(****************************************************************Mode 21 : Mode alerte préparateur****************************************************************)
Mode_21 := Numero_Mode = 21 AND Enable;
TON_Mode21(IN:=(Mode_21 AND NOT Fin_Action), PT:= T#10s);
IF(Mode_21)
	THEN
	(*Gestion du texte du mode*)
	Out_Texte_FR := 'ALERTE PREPARATEUR';
	Out_Texte_ENG := 'PREPARATOR ALERT';

	(*Initialisation des actionneurs non utilisés*)
	Cmd_Douche := FALSE;
	Cmd_Lavabo := FALSE;
	Cmd_Douchette := FALSE;
	Cmd_NEP := FALSE;
	Cmd_Electrovanne_Douche := FALSE;
	Cmd_Electrovanne_Lavabo := FALSE;
	Cmd_Verin_WC_GV := FALSE;
	Cmd_Verin_WC_PV := FALSE;
END_IF;

(****************************************************************Mode 22 : Mode alerte évaluateur****************************************************************)
Mode_22 := Numero_Mode = 22 AND Enable;
TON_Mode22(IN:=(Mode_22 AND NOT Fin_Action), PT:= T#10s);
IF(Mode_22)
	THEN
	(*Gestion du texte du mode*)
	Out_Texte_FR := 'ALERTE EVALUATEUR';
	Out_Texte_ENG := 'EVALUATOR ALERT';

	(*Initialisation des actionneurs non utilisés*)
	Cmd_Douche := FALSE;
	Cmd_Lavabo := FALSE;
	Cmd_Douchette := FALSE;
	Cmd_NEP := FALSE;
	Cmd_Electrovanne_Douche := FALSE;
	Cmd_Electrovanne_Lavabo := FALSE;
	Cmd_Verin_WC_GV := FALSE;
	Cmd_Verin_WC_PV := FALSE;
END_IF;

(****************************************************************Mode 23 : Mode évaluation (sans moteur bypass)****************************************************************)
Mode_23 := Numero_Mode = 23 AND Enable;
F_TRIG_Texte23(CLK:= (Valid_Texte AND Mode_23));
IF(Mode_23)
	THEN
	(*Gestion du texte du mode*)
	Out_Texte_FR := 'EVALUATION';
	Out_Texte_ENG := 'EVALUATION';

	(*Gestion des lectures consignes du mode*)
	Out_Debit_Souf 			:= Cons_Deb_Soufflage;
	Out_Debit_Ext 			:= Cons_Deb_Extraction;
	Out_Temp_Eau 			:= Cons_Temperature_Eau;

	(*Initialisation des actionneurs non utilisés*)
	Cmd_Douche := FALSE;
	Cmd_Lavabo := FALSE;
	Cmd_Douchette := FALSE;
	Cmd_NEP := FALSE;
	Cmd_Vidange_Douche := FALSE;
	//Cmd_Vidange_Lavabo := FALSE;
	Cmd_Electrovanne_Douche := FALSE;
	Cmd_Electrovanne_Lavabo := FALSE;
	Cmd_Prise := FALSE;
	Cmd_Verin_WC_GV := FALSE;
	Cmd_Verin_WC_PV := FALSE;
END_IF;

(****************************************************************Mode 24 : Mode évaluation (avec moteur bypass)****************************************************************)
Mode_24 := Numero_Mode = 24 AND Enable;
F_TRIG_Texte24(CLK:= (Valid_Texte AND Mode_24));
IF(Mode_24)
	THEN
	(*Gestion du texte du mode*)
	Out_Texte_FR := 'EVALUATION AVEC AIR';
	Out_Texte_ENG := 'EVALUATION WITH AIR FLOW';

	(*Gestion des lectures consignes du mode*)
	Out_Debit_Souf 			:= 0.0;
	Out_Debit_Ext 			:= 0.0;
	Out_Temp_Eau 			:= Cons_Temperature_Eau;
	Out_Cons_Moteur_ByPass := REAL_TO_INT(Cons_Moteur_ByPass);

	(*Initialisation des actionneurs non utilisés*)
	Cmd_Douche := FALSE;
	Cmd_Lavabo := FALSE;
	Cmd_Douchette := FALSE;
	Cmd_NEP := FALSE;
	Cmd_Vidange_Douche := FALSE;
	Cmd_Vidange_Lavabo := FALSE;
	Cmd_Electrovanne_Douche := FALSE;
	Cmd_Electrovanne_Lavabo := FALSE;
	Cmd_Prise := FALSE;
	Cmd_Verin_WC_GV := FALSE;
	Cmd_Verin_WC_PV := FALSE;
	ELSE
	Out_Cons_Moteur_ByPass := 0;
END_IF;

(****************************************************************Mode 25 : Mode Mise en condition****************************************************************)
Mode_25 := Numero_Mode = 25 AND Enable;
F_TRIG_Mode25(CLK:= ((Valid_Texte OR R_TRIG_Valide_TempHygro.Q) AND Mode_25));
IF(Mode_25  AND NOT Fin_Action)
THEN
	(*Gestion du texte du mode*)
	Out_Texte_FR := 'MISE EN CONDITION';
	Out_Texte_ENG := 'CONDITIONING BOOTH';
	
	(*Initialisation des actionneurs non utilisés*)
	Cmd_Douche := FALSE;
	Cmd_Lavabo := FALSE;
	Cmd_Douchette := FALSE;
	Cmd_NEP := FALSE;
	Cmd_Vidange_Douche := FALSE;
	//Cmd_Vidange_Lavabo := FALSE;
	Cmd_Electrovanne_Douche := FALSE;
	Cmd_Electrovanne_Lavabo := FALSE;
	Cmd_Prise := FALSE;
	Cmd_Verin_WC_GV := FALSE;
	Cmd_Verin_WC_PV := FALSE;
	
	(*Gestion des lectures consignes du mode*)
	Out_Debit_Souf 			:= Cons_Deb_Soufflage;
	Out_Debit_Ext 			:= Cons_Deb_Extraction;
	Out_Para_11				:= Cons_Para_11;
	Out_Para_12				:= Cons_Para_12;
END_IF;
(*Validation de la régulation de la température pour passer en mode 13*)
(*Température*)
IF ((S_Ecart_Regul_PID_Temp >= 0.0) AND (S_Ecart_Regul_PID_Temp <= 2.0) AND Mode_25) THEN Temp_Ok := TRUE; ELSE Temp_Ok := FALSE; END_IF;
TON_Temp_Ok(IN:= Temp_Ok, PT:= T#15M);
(*Hygrométrie*)
IF ((S_Ecart_Regul_PID_Hygro >= 0.0) AND (S_Ecart_Regul_PID_Hygro <= 5.0) AND Mode_25) THEN Hygro_Ok := TRUE; ELSE Hygro_Ok := FALSE; END_IF;
TON_Hygro_Ok(IN:= Hygro_Ok, PT:= T#15M);
Validation_Temp_Hygro := TON_Temp_Ok.Q AND TON_Hygro_Ok.Q;
R_TRIG_Valide_TempHygro(CLK:= Validation_Temp_Hygro);

(*TP_RAZ_Mode25(IN:= Validation_Temp_Hygro, PT:= T#1s);
Validation_Temp_Hygro := (SEL(Validation_Temp_Hygro, Validation_Temp_Hygro, FALSE) OR TP_RAZ_Mode25.Q);*)

(****************************************************************Mode 26 : Mode chasse d'eau petit volume****************************************************************)
Mode_26 := Numero_Mode = 26 AND Enable;
IF(Mode_26 AND NOT Fin_Action)
	THEN
	(*Gestion du texte*)
	Out_Texte_FR := 'CHASSE D EAU PETIT VOLUME';
	Out_Texte_ENG := 'SMALL VOLUME TOILET FLUSH';

	(*Gestion du décompte de la temporisation du mode*)
	Out_Restant_Seconde := TON_Mode26.Seconde_Restant;
	Out_Restant_Minute := TON_Mode26.Minute_Restant;
	Out_Restant_Heure := TON_Mode26.Heure_Restant;

	(*Démarrage du premier cycle de chasse avant la temporisation*)
	R_TRIG_Cpt_Chasse_PV(CLK:= (Mode_26));

	(*Comptage du nombre de cycle x*)
	IF (TON_Mode26.Q OR R_TRIG_Cpt_Chasse_PV.Q)
		THEN
		Cpt_Chasse_PV := Cpt_Chasse_PV + 1;
		Restart_Chasse_PV := TRUE;
	END_IF;

	(*Initialisation des actionneurs non utilisés*)
	Cmd_Douche := FALSE;
	Cmd_Lavabo := FALSE;
	Cmd_Douchette := FALSE;
	Cmd_NEP := FALSE;
	Cmd_Electrovanne_Douche := FALSE;
	Cmd_Electrovanne_Lavabo := FALSE;
	Cmd_Prise := FALSE;
	Cmd_Verin_WC_GV := FALSE;
END_IF;
(*************************************Temporisation du décompte du mode*************************************)
TON_Mode26(
	Enable:= ((Mode_26 OR Comande_Pause OR Tp_ChasseEau_PV.Q) AND NOT Restart_Chasse_PV),
	Pause:= Comande_Pause OR Tp_ChasseEau_PV.Q,
	In_Cons_Seconde:= Tempo_Transition_Seconde,
	In_Cons_Minute:= Tempo_Transition_Minute,
	In_Cons_Heure:= Tempo_Transition_Heure);
Restart_Chasse_PV := FALSE;
(*Commande de la chasse d'eau pendant x secondes*)
Tp_ChasseEau_PV(IN:= TON_Mode26.Q OR R_TRIG_Cpt_Chasse_PV.Q, PT:= T#2s);
IF (Tp_ChasseEau_PV.Q AND Mode_26) THEN Cmd_Verin_WC_PV := TRUE; ELSE Cmd_Verin_WC_PV := FALSE; END_IF;
(*FIn du mode quand le nombre de cycle est atteint*)
IF ((Cpt_Chasse_PV >= Cons_Nbre_Chasse) AND Mode_26 AND NOT Tp_ChasseEau_PV.Q)
	THEN Etp_Suiv_ChasseEau_PV := TRUE; Cpt_Chasse_PV := 0.0;
	ELSE Etp_Suiv_ChasseEau_PV := FALSE; END_IF;
	
(****************************************************************Mode 27 : Mode lavage NEP ****************************************************************)
Mode_27 := Numero_Mode = 27 AND Enable;
IF(Mode_27  AND NOT Fin_Action)
	THEN
	(*Gestion du texte*)
	IF(E_Vanne_Vidange_Douche_Ouv)
		THEN
		Out_Texte_FR := 'LAVAGE NEP';
		Out_Texte_ENG := 'CLEANING';
		ELSE
		Out_Texte_FR := 'LAVAGE NEP - OUVERTURE BONDE';
		Out_Texte_ENG :=  'CLEANING - OPENING DRAIN';
	END_IF;
	IF(RS_Fin_Mode_27.Q1)
		THEN
		Out_Texte_FR := 'LAVAGE NEP - ARRET LAVAGE';
		Out_Texte_ENG := 'CLEANING - STOPING CLEANING';
	END_IF;

	(*Gestion de la commande de la NEP et de la vidange*)
	Cmd_Vidange_Douche := TRUE;
	
	IF( RS_Fin_Mode_27.Q1)
		THEN
		Out_Restant_Seconde := 0.0;
		Out_Restant_Minute := 0.0;
		Out_Restant_Heure := 0.0;
		Cmd_NEP := FALSE;
		ELSE
		IF(E_Vanne_Vidange_Douche_Ouv)
			THEN
			Cmd_NEP := TRUE;
			ELSE
			Cmd_NEP := FALSE;
		END_IF;
	END_IF;

	(*Gestion de la commande pause*)
	IF(Comande_Pause)
		THEN
		Cmd_NEP := FALSE;
	END_IF;

	(*Gestion du décompte de la temporisation du mode*)
	Out_Restant_Seconde := TON_Mode27.Seconde_Restant;
	Out_Restant_Minute := TON_Mode27.Minute_Restant;
	Out_Restant_Heure := TON_Mode27.Heure_Restant;

	(*Gestion des lectures consignes du mode*)
	Out_Debit_Souf 			:= Cons_Deb_Soufflage;
	Out_Debit_Ext 			:= Cons_Deb_Extraction;
	(*Out_Temp_Eau 			:= Cons_Temperature_Eau;*)

	(*Initialisation des actionneurs non utilisés*)
	Cmd_Douche := FALSE;
	Cmd_Lavabo := FALSE;
	Cmd_Douchette := FALSE;
	Cmd_Vidange_Lavabo := FALSE;
	Cmd_Electrovanne_Douche := FALSE;
	Cmd_Electrovanne_Lavabo := FALSE;
	Cmd_Prise := FALSE;
	Cmd_Verin_WC_GV := FALSE;
	Cmd_Verin_WC_PV := FALSE;
END_IF;
(*************************************Temporisation du décompte du mode*************************************)
TON_Mode27(
Enable:= (Mode_27 AND ((E_Vanne_Vidange_Douche_Ouv AND E_Vanne_Alim_NEP_Ouv) OR Comande_Pause)),
Pause:= Comande_Pause,
In_Cons_Seconde:= Tempo_Transition_Seconde,
In_Cons_Minute:= Tempo_Transition_Minute,
In_Cons_Heure:= Tempo_Transition_Heure);

(*Activation de la fin du mode*)
RS_Fin_Mode_27(SET:= TON_Mode27.Q, RESET1:= NOT Mode_27);
IF( RS_Fin_Mode_27.Q1)
	THEN
	Out_Restant_Seconde := 0.0;
	Out_Restant_Minute := 0.0;
	Out_Restant_Heure := 0.0;
END_IF;

(****************************************************************Mode 28 : Mode en fonctionnement****************************************************************)
Mode_28 := Numero_Mode = 28 AND Enable;
F_TRIG_Mode28(CLK:= (Valid_Texte AND Mode_28));
IF(Mode_28 AND NOT Fin_Action)
THEN
	(*Gestion du texte du mode*)
	Out_Texte_FR := 'CABINE EN CONDITION';
	Out_Texte_ENG := 'BOOTH IN CONDITION';
	
	(*Initialisation des actionneurs non utilisés*)
	Cmd_Douche := FALSE;
	Cmd_Lavabo := FALSE;
	Cmd_Douchette := FALSE;
	Cmd_NEP := FALSE;
	Cmd_Vidange_Douche := FALSE;
	//Cmd_Vidange_Lavabo := FALSE;
	Cmd_Electrovanne_Douche := FALSE;
	Cmd_Electrovanne_Lavabo := FALSE;
	Cmd_Prise := FALSE;
	Cmd_Verin_WC_GV := FALSE;
	Cmd_Verin_WC_PV := FALSE;
	
	(*Gestion des lectures consignes du mode*)
	Out_Debit_Souf 			:= Cons_Deb_Soufflage;
	Out_Debit_Ext 			:= Cons_Deb_Extraction;
	Out_Para_11				:= Cons_Para_11;
	Out_Para_12				:= Cons_Para_12;
END_IF;

(****************************************************************Mode 30 à 59 : Mode Texte 1 à 30****************************************************************)
Mode_30 := ((Numero_Mode >= 30) AND (Numero_Mode <= 59)) AND Enable;
F_TRIG_Texte30(CLK:= (Valid_Texte AND Mode_30));
IF(Mode_30)
THEN
	(*Gestion du texte du mode*)
	Out_Texte_FR := Tab_Mode_Texte[1, (REAL_TO_INT(Numero_Mode))];
	Out_Texte_ENG := Tab_Mode_Texte[2, (REAL_TO_INT(Numero_Mode))];

	(*Initialisation des actionneurs non utilisés*)
	Cmd_Douche := FALSE;
	Cmd_Lavabo := FALSE;
	Cmd_Douchette := FALSE;
	Cmd_NEP := FALSE;
	Cmd_Electrovanne_Douche := FALSE;
	Cmd_Electrovanne_Lavabo := FALSE;
	Cmd_Verin_WC_GV := FALSE;
	Cmd_Verin_WC_PV := FALSE;
END_IF;

(****************************************************************Mode 99 : Mode END****************************************************************)
IF(Numero_Mode = 99 AND Enable)
	THEN
	Mode_END := TRUE;
	ELSE
	Mode_END := FALSE;
END_IF;

(****************************************************************Sécurité de débordement de la douche****************************************************************)
(*Sécurité douche version temporisation pour le mode 2*)
Temp_Secu_Douche := TO_TIME((TO_DINT(Temp_Secu_Debord_Douche + 5)) * 1000);
Temp_Secu_Debord_Douche_Int := (Temp_Secu_Debord_Douche); (*Pour lecture IHM*)
TON_Secu_Douche(IN:= ((Mode_2 AND (Cmd_Douche OR Cmd_Electrovanne_Douche)) AND NOT Cmd_Vidange_Douche), PT:= Temp_Secu_Douche);
IF(TON_Secu_Douche.Q)
	THEN
	Securite_Debord_Douche := TRUE;
	Cmd_Douche := FALSE;
	ELSE
	Securite_Debord_Douche := FALSE;
END_IF;

(*Sécurité lavabo version temporisation pour le mode 5*)
Temp_Secu_Lavabo := TO_TIME((TO_DINT(Temp_Secu_Debord_Lavabo + 5)) * 1000);
Temp_Secu_Debord_Lavabo_Int := (Temp_Secu_Debord_Lavabo); (*Pour lecture IHM*)
TON_Secu_Lavabo(IN:= ((Mode_5 AND (Cmd_Lavabo OR Cmd_Electrovanne_Lavabo)) AND NOT Cmd_Vidange_Lavabo) , PT:= Temp_Secu_Lavabo);
IF(TON_Secu_Lavabo.Q)
	THEN
	Securite_Debord_Lavabo := TRUE;
	Cmd_Lavabo := FALSE;
	ELSE
	Securite_Debord_Lavabo := FALSE;
END_IF;

(*Sécurité douche version débitmétre pour le mode 13*)
Secu_Volume_Douche := (((Cmd_Electrovanne_Douche AND Option_Debitmetre_Douche) AND NOT Cmd_Vidange_Douche)
						AND (Out_Volume_Eau_Douche > Volume_Secu_Debord_Douche + 0.5));
IF(Mode_13 AND Secu_Volume_Douche)
	THEN
	Securite_Debord_Douche_Debit := TRUE;
	Cmd_Electrovanne_Douche := FALSE;
	ELSE
	Securite_Debord_Douche_Debit := FALSE;
END_IF;

(*Sécurité lavabo version débitmétre pour le mode 15*)
Secu_Volume_Lavabo := (((Cmd_Electrovanne_Lavabo AND Option_Debitmetre_Lavabo) AND NOT Cmd_Vidange_Lavabo)
						AND (Out_Volume_Eau_Lavabo > Volume_Secu_Debord_Lavabo + 0.5));
IF(Mode_15 AND Secu_Volume_Lavabo)
	THEN
	Securite_Debord_Lavabo_Debit := TRUE;
	Cmd_Electrovanne_Lavabo := FALSE;
	ELSE
	Securite_Debord_Lavabo_Debit := FALSE;
END_IF;

(****************************************************************Gestion initialisation des variables****************************************************************)
IF(Numero_Mode = 0 OR Numero_Etape = 0)
	THEN
	(*Initialisation des actionneurs*)
	Cmd_Douche := FALSE;
	Cmd_Lavabo := FALSE;
	Cmd_Douchette := FALSE;
	Cmd_NEP := FALSE;
	Cmd_Vidange_Douche := FALSE;
	Cmd_Vidange_Lavabo := FALSE;
	Cmd_Electrovanne_Douche := FALSE;
	Cmd_Electrovanne_Lavabo := FALSE;
	Cmd_Prise := FALSE;
	Cmd_Verin_WC_GV := FALSE;
	Cmd_Verin_WC_PV := FALSE;

	Out_Restant_Seconde := 0.0;
	Out_Restant_Minute := 0.0;
	Out_Restant_Heure := 0.0;

	Out_Volume_Eau_Douche := 0.0;
	Out_Volume_Eau_Lavabo := 0.0;
	Out_Debit_Souf := 0.0;
	Out_Debit_Ext := 0.0;
	Out_Temp_Eau := 0.0;
	Out_Cons_V3V_Eau_Mitig := 0.0;
	Cpt_Chasse_GV := 0.0;
	Restart_Chasse_GV := FALSE;
	Etp_Suiv_ChasseEau_GV := FALSE;
	Cpt_Chasse_PV := 0.0;
	Restart_Chasse_PV := FALSE;
	Etp_Suiv_ChasseEau_PV := FALSE;
	Out_Para_11 := 0.0;
	Out_Para_12 := 0.0;
	Out_Para_13 := 0.0;
	Out_Para_14 := 0.0;
	Out_Para_15 := 0.0;

	Out_Texte_FR := '';
	Out_Texte_ENG := '';

	R_TRIG_Mode12(CLK := FALSE);
	Integr_Vol_Eau_Mode12(Enable:= FALSE);
	R_TRIG_Mode13(CLK := FALSE);
	Integr_Vol_Eau_Mode13(Enable:= FALSE);
	R_TRIG_Mode14(CLK := FALSE);
	Integr_Vol_Eau_Mode14(Enable:= FALSE);
	R_TRIG_Mode15(CLK := FALSE);
	Integr_Vol_Eau_Mode15(Enable:= FALSE);
	R_TRIG_Cpt_Chasse_GV(CLK:= FALSE);
	R_TRIG_Cpt_Chasse_PV(CLK:= FALSE);

	TON_Temp_Ok(IN:= FALSE);
	TON_Hygro_Ok(IN:= FALSE);
	TP_RAZ_Mode25(IN:= FALSE);
	F_TRIG_Mode25(CLK:= FALSE);
	F_TRIG_Mode28(CLK:= FALSE);
	Temp_Ok := FALSE;
	Hygro_Ok := FALSE;
	Validation_Temp_Hygro := FALSE;
END_IF;

(****************************************************************Gestion du passage entre chaque mode****************************************************************)
				(*Mode temporisé*)
Fin_Action := 		(RS_Fin_Mode_1.Q1 AND (E_Vanne_Alim_Douche_Ferm OR Option_Debitmetre_Douche)) (*Mode douche avec vidange*)
				OR ((RS_Fin_Mode_2.Q1 AND (E_Vanne_Alim_Douche_Ferm OR Option_Debitmetre_Douche) OR Securite_Debord_Douche)) (*Mode douche sans vidange*)
				OR (RS_Fin_Mode_4.Q1 AND (E_Vanne_Alim_Lavabo_Ferm OR Option_Debitmetre_Lavabo)) (*Mode lavabo avec vidange*)
				OR ((RS_Fin_Mode_5.Q1 AND (E_Vanne_Alim_Lavabo_Ferm OR Option_Debitmetre_Lavabo) OR Securite_Debord_Lavabo)) (*Mode lavabo sans vidange*)
				OR (RS_Fin_Mode_7.Q1) (*Mode vidange*)
				OR (RS_Fin_Mode_18.Q1 AND E_Vanne_Alim_NEP_Ferm) (*Mode lavage eau chaude*)
				OR (RS_Fin_Mode_19.Q1 AND E_Vanne_Alim_NEP_Ferm) (*Mode lavage eau froide*)
				OR (RS_Fin_Mode_27.Q1 AND E_Vanne_Alim_NEP_Ferm) (*Mode lavage*)
				(*Mode Gestion volume*)
				OR R_TRIG_Mode12.Q OR R_TRIG_Mode13.Q OR R_TRIG_Mode14.Q OR R_TRIG_Mode15.Q
				 (*Gestion des modes sans validation*)
				OR TON_Mode8.Q OR TON_Mode22.Q OR TON_Mode21.Q OR TON_Mode10.Q OR TON_Mode6.Q OR TON_Mode11.Q
				(*Mode texte*)
				OR F_TRIG_Texte3.Q OR F_TRIG_Texte23.Q OR F_TRIG_Texte30.Q OR F_TRIG_Texte16.Q OR F_TRIG_Texte17.Q OR F_TRIG_Texte24.Q
				(*Mode chasse d'eau*)
				OR Etp_Suiv_ChasseEau_GV OR Etp_Suiv_ChasseEau_PV
				(*Mode pour enceintes climatiques*)
				OR F_TRIG_Mode25.Q OR F_TRIG_Mode28.Q;

END_FUNCTION_BLOCK

// ---- POUs/Block/Cabines/Integr_Vol_Eau.TcPOU
FUNCTION_BLOCK Integr_Vol_Eau
VAR_INPUT
	Enable :BOOL;
	Mes_Debit_Eau :REAL; (*Mesure débit en l/min*)
END_VAR
VAR_OUTPUT
	Volume_Eau :REAL; (*Volume d'eau en Litre*)
END_VAR
VAR
	TON_Inc: TON;
	R_TRIG_1	:R_TRIG;
	R_TRIG_Inc: R_TRIG;
	TOP_INTEGRATION	:BOOL;
	Reset	:BOOL;

	FlowRate_MPS :REAL; (*Debit d'eau en l/s*)
	TimeElapsed :TIME; (*Temps écoulé depuis la dernière mesur*)
END_VAR

(*Comptage des secondes*)
TON_Inc(IN:= (NOT TOP_INTEGRATION AND NOT Reset), PT:= T#1s, Q=> TOP_INTEGRATION );
R_TRIG_Inc(CLK:= TOP_INTEGRATION);

R_TRIG_1(CLK:=TOP_INTEGRATION);
Reset := NOT Enable;

(*Convertion du débit d'eau l/min en l/s*)
FlowRate_MPS := Mes_Debit_Eau / 60.0;

(*Condition d'activation : mettre la variable Enbale à TRUE pour exécuter le calcul*)
IF (TOP_INTEGRATION)
	THEN
	Volume_Eau			:= Volume_Eau + FlowRate_MPS;
END_IF;

Volume_Eau:=SEL(Reset,(Volume_Eau),0.0);
Mes_Debit_Eau:=SEL(Reset,Mes_Debit_Eau,0.0);

END_FUNCTION_BLOCK

// ---- POUs/Block/Autres/Prise.TcPOU
FUNCTION_BLOCK Prise
VAR_INPUT
	Enable:						BOOL;
	Cmd_Prise:					BOOL;	(*Commande de la prise de courant*)
	Cabine_Seche: 				BOOL;
	Statut_Ferm_Reg_Douche:		BOOL;	(*Statut fermeture du registre de la vanne de la douche / 1 = Fermé / si registre non présence forcer la variable à TRUE*)
	Statut_Ferm_Lavabo:			BOOL;	(*Statut fermeture du registre de la vanne du lavabo / 1 = Fermé / si registre non présence forcer la variable à TRUE*)
	Statut_Electrovanne_Douche:		BOOL;
	Statut_Electrovanne_Lavabo:		BOOL;
	Statut_Def_Prise_Porte_Ouverte:		BOOL;
	Statut_Def_Discord_Alim_Prise:		BOOL;
	Statut_Defaut_Discord_PC_Cab:		BOOL;
END_VAR
VAR_OUTPUT
	STOR_Prise:			BOOL;			(*Commande de la sortie TOR de la prise*)
END_VAR
VAR
END_VAR

IF(Enable AND Cmd_Prise
	AND (Statut_Ferm_Reg_Douche OR Cabine_Seche OR Option_Debitmetre_Lavabo) AND (Statut_Ferm_Lavabo OR Cabine_Seche OR Option_Debitmetre_Lavabo)
	AND ( NOT Statut_Electrovanne_Douche OR Cabine_Seche) AND (NOT Statut_Electrovanne_Lavabo OR Cabine_Seche)
	AND NOT Statut_Def_Prise_Porte_Ouverte AND NOT Statut_Def_Discord_Alim_Prise AND NOT Statut_Defaut_Discord_PC_Cab)
	THEN
		STOR_Prise := TRUE;
	ELSE
		STOR_Prise := FALSE;
END_IF;

END_FUNCTION_BLOCK

// ---- POUs/h_Enr_Recette.TcPOU
PROGRAM h_Enr_Recette
VAR
	i: INT;
	F_TRIG_Reset: F_TRIG;
	j: INT;
	R_TRIG_Enr: R_TRIG;
END_VAR

R_TRIG_Enr(CLK:= Cmd_Enr_Recette AND NOT Mode_Cabine_Automatique AND NOT Validation_Recette_Auto AND NOT Start_Recette_Mode_Auto);
IF(R_TRIG_Enr.Q)
	THEN
	(*Transfert dans la recette à enregistrée dans le tableau recette automatique*)
	FOR i := 1 TO 29 BY 1 DO
		Tab_Recette_Auto[Numero_Recette_Sel, i, 1] := Tab_Enr_Recette[0, i, 1];
		Tab_Recette_Auto[Numero_Recette_Sel, i, 2] := Tab_Enr_Recette[0, i, 2];
		Tab_Recette_Auto[Numero_Recette_Sel, i, 3] := Tab_Enr_Recette[0, i, 3];
		Tab_Recette_Auto[Numero_Recette_Sel, i, 4] := Tab_Enr_Recette[0, i, 4];
		Tab_Recette_Auto[Numero_Recette_Sel, i, 5] := Tab_Enr_Recette[0, i, 5];
		Tab_Recette_Auto[Numero_Recette_Sel, i, 6] := Tab_Enr_Recette[0, i, 6];
		Tab_Recette_Auto[Numero_Recette_Sel, i, 7] := Tab_Enr_Recette[0, i, 7];
		Tab_Recette_Auto[Numero_Recette_Sel, i, 8] := Tab_Enr_Recette[0, i, 8];
		Tab_Recette_Auto[Numero_Recette_Sel, i, 9] := Tab_Enr_Recette[0, i, 9];
		Tab_Recette_Auto[Numero_Recette_Sel, i, 10] := Tab_Enr_Recette[0, i, 10];
		Tab_Recette_Auto[Numero_Recette_Sel, i, 11] := Tab_Enr_Recette[0, i, 11];
		Tab_Recette_Auto[Numero_Recette_Sel, i, 12] := Tab_Enr_Recette[0, i, 12];
		Tab_Recette_Auto[Numero_Recette_Sel, i, 13] := Tab_Enr_Recette[0, i, 13];
		Tab_Recette_Auto[Numero_Recette_Sel, i, 14] := Tab_Enr_Recette[0, i, 14];
		Tab_Recette_Auto[Numero_Recette_Sel, i, 15] := Tab_Enr_Recette[0, i, 15];
	END_FOR;
END_IF;
(*Reset du tableau sur le front descendant*)
F_TRIG_Reset(CLK:= Cmd_Enr_Recette);
IF(F_TRIG_Reset.Q)
	THEN
	FOR j := 1 TO 29 BY 1 DO
		Tab_Enr_Recette[0, j, 1] := 0;
		Tab_Enr_Recette[0, j, 2] := 0;
		Tab_Enr_Recette[0, j, 3] := 0;
		Tab_Enr_Recette[0, j, 4] := 0;
		Tab_Enr_Recette[0, j, 5] := 0;
		Tab_Enr_Recette[0, j, 6] := 0;
		Tab_Enr_Recette[0, j, 7] := 0;
		Tab_Enr_Recette[0, j, 8] := 0;
		Tab_Enr_Recette[0, j, 9] := 0;
		Tab_Enr_Recette[0, j, 10] := 0;
		Tab_Enr_Recette[0, j, 11] := 0;
		Tab_Enr_Recette[0, j, 12] := 0;
		Tab_Enr_Recette[0, j, 13] := 0;
		Tab_Enr_Recette[0, j, 14] := 0;
		Tab_Enr_Recette[0, j, 15] := 0;
	END_FOR;
	ELSE
	j := 1;
END_IF;

END_PROGRAM

// ---- POUs/i_Protocol_Auto.TcPOU
PROGRAM i_Protocol_Auto
VAR
(*Validation de la recette sélectionnée*)
	n: INT;
	i: INT;
	R_TRIG_RAZ_etape: R_TRIG;
(*initialisation des valeurs*)
	j: INT;
(*Execution de la recette en mode auto*)
	R_TRIG_Dem: R_TRIG;
	R_TRIG1: R_TRIG;
(*Gestion de la poste de ventilation*)
	F_TRIG_Fin_Post_Ventil: F_TRIG;
	TON_PV: TON;
	R_TRIG_PV: R_TRIG;
END_VAR

(*MEMSET(ADR(Tab_Nom_Recette),0,SIZEOF(Tab_Nom_Recette));
MEMSET(ADR(Tab_Mode_Texte),0,SIZEOF(Tab_Mode_Texte));*)

(************************************************************************************************************************Gestion Arrêt du grafcet*)
Mode_Arret_Auto := 	(Reset_Mode_Auto(*Fin de la recette*)
					OR ((Numero_Mode_Auto = 1) AND Mode_Auto.Mode_END) (*Fin de la recette*)
					OR (Mode_Auto.Mode_12 AND Defaut_Discord_Deb_Eau_Douche)
					OR (Mode_Auto.Mode_13 AND Defaut_Discord_Deb_Eau_Douche)
					OR (Mode_Auto.Mode_14 AND Defaut_Discord_Deb_Eau_Lavabo)
					OR (Mode_Auto.Mode_15 AND Defaut_Discord_Deb_Eau_Lavabo)
					OR Defaut_Debordement_Douche OR Defaut_Debordement_Lavabo)
					OR (Mode_Auto.Mode_4 AND Defaut_Discord_Deb_Eau_Lavabo AND Option_Debitmetre_Lavabo)
					OR (Mode_Auto.Mode_5 AND Defaut_Discord_Deb_Eau_Lavabo AND Option_Debitmetre_Lavabo)
					OR (Mode_Auto.Mode_1 AND Defaut_Discord_Deb_Eau_Douche AND Option_Debitmetre_Douche)
					OR (Mode_Auto.Mode_2 AND Defaut_Discord_Deb_Eau_Douche AND Option_Debitmetre_Douche)
					OR (RS_MEnCond.Q1 AND Defaut_Arret_Mode25 AND Option_Cabine_Climatique) //RS_MEnCond.Q1 Correspond au démarrage de la CTA durant une recette
					OR Defaut_Discord_Reg_Etanche_Ext OR Defaut_Sonde_Temp_Eau_Mitig;

(************************************************************************************************************************Validation de la recette sélectionnée*)
IF(Validation_Recette_Auto AND NOT Mode_Arret_Auto)
	THEN
	(*Remise à zéro du nombre d'étape total avant le calcul du nombre d'étape total*)
	R_TRIG_RAZ_etape(CLK:= Validation_Recette_Auto);
	IF (R_TRIG_RAZ_etape.Q) THEN Nbre_Etape_Totale := 0; END_IF;
	(*Transfert dans la recette 0 de la recettte sélectionnée*)
	FOR i := 1 TO 29 BY 1 DO
		Tab_Recette_Auto[0, i, 1] := Tab_Recette_Auto[Numero_Recette_Sel, i, 1];
		Tab_Recette_Auto[0, i, 2] := Tab_Recette_Auto[Numero_Recette_Sel, i, 2];
		Tab_Recette_Auto[0, i, 3] := Tab_Recette_Auto[Numero_Recette_Sel, i, 3];
		Tab_Recette_Auto[0, i, 4] := Tab_Recette_Auto[Numero_Recette_Sel, i, 4];
		Tab_Recette_Auto[0, i, 5] := Tab_Recette_Auto[Numero_Recette_Sel, i, 5];
		Tab_Recette_Auto[0, i, 6] := Tab_Recette_Auto[Numero_Recette_Sel, i, 6];
		Tab_Recette_Auto[0, i, 7] := Tab_Recette_Auto[Numero_Recette_Sel, i, 7];
		Tab_Recette_Auto[0, i, 8] := Tab_Recette_Auto[Numero_Recette_Sel, i, 8];
		Tab_Recette_Auto[0, i, 9] := Tab_Recette_Auto[Numero_Recette_Sel, i, 9];
		Tab_Recette_Auto[0, i, 10] := Tab_Recette_Auto[Numero_Recette_Sel, i, 10];
		Tab_Recette_Auto[0, i, 11] := Tab_Recette_Auto[Numero_Recette_Sel, i, 11];
		Tab_Recette_Auto[0, i, 12] := Tab_Recette_Auto[Numero_Recette_Sel, i, 12];
		Tab_Recette_Auto[0, i, 13] := Tab_Recette_Auto[Numero_Recette_Sel, i, 13];
		Tab_Recette_Auto[0, i, 14] := Tab_Recette_Auto[Numero_Recette_Sel, i, 14];
		Tab_Recette_Auto[0, i, 15] := Tab_Recette_Auto[Numero_Recette_Sel, i, 15];
	END_FOR;
	(*Calcul etape total*)
	FOR n := 1 TO 29 BY 1 DO
		IF(Tab_Recette_Auto[Numero_Recette_Sel, n, 1] = 99)
			THEN
			Nbre_Etape_Totale := n - 1;
			n := 29;
		END_IF;
	END_FOR;
	ELSE;
	R_TRIG_RAZ_etape(CLK:= FALSE);
	i := 0;
	n := 0;
END_IF;

(************************************************************************************************************************Démarrage du mode auto*)
IF(Mode_Cabine_Automatique AND (Numero_Mode_Auto = 0) AND NOT Mode_Arret_Auto)
	THEN
	Numero_Mode_Auto := 1;
END_IF;

(*Gestion du case du mode auto*)
CASE Numero_Mode_Auto OF
(*******************************************************************************************Etape 0 : Attente*)
0:
j:=0; (*Initlisation de la variable boucle FOR d'initialisation*)
Mode_Auto(
	Enable:= 					(FALSE),
	Numero_Etape:= 				Numero_Etape_Actuel);

(*******************************************************************************************Etape 1 :Execution de la recette en mode auto*)
1:
R_TRIG_Dem(CLK:= (Numero_Mode_Auto = 1));
(*Démarrage de l'étape 1 de la recette*)
IF(R_TRIG_Dem.Q)
	THEN
	Numero_Etape_Actuel := Numero_Etape_Actuel + 1;
END_IF;

(*Bloc fontion recette*)
Mode_Auto(
	Enable:= 					(Numero_Mode_Auto = 1),
	Numero_Etape:= 				Numero_Etape_Actuel,
	Numero_Mode:= 				Tab_Recette_Auto[0, LIMIT(1,Numero_Etape_Actuel,30), 1],
	Tempo_Transition_seconde:=	Tab_Recette_Auto[0, LIMIT(1,Numero_Etape_Actuel,30), 2],
	Tempo_Transition_Minute:=	Tab_Recette_Auto[0, LIMIT(1,Numero_Etape_Actuel,30), 3],
	Tempo_Transition_Heure:= 	Tab_Recette_Auto[0, LIMIT(1,Numero_Etape_Actuel,30), 4],
	Cons_Volume_Eau_Douche:= 	Tab_Recette_Auto[0, LIMIT(1,Numero_Etape_Actuel,30), 6],
	Cons_Volume_Eau_Lavabo:=	Tab_Recette_Auto[0, LIMIT(1,Numero_Etape_Actuel,30), 6],
	Cons_Deb_Soufflage:= 		Tab_Recette_Auto[0, LIMIT(1,Numero_Etape_Actuel,30), 7],
	Cons_Deb_Extraction:=		Tab_Recette_Auto[0, LIMIT(1,Numero_Etape_Actuel,30), 8],
	Cons_Temperature_Eau:= 		Tab_Recette_Auto[0, LIMIT(1,Numero_Etape_Actuel,30), 9],
	Cons_Nbre_Chasse:= 			Tab_Recette_Auto[0, LIMIT(1,Numero_Etape_Actuel,30), 10],
	Cons_Para_11:= 				Tab_Recette_Auto[0, LIMIT(1,Numero_Etape_Actuel,30), 11],
	Cons_Para_12:= 				Tab_Recette_Auto[0, LIMIT(1,Numero_Etape_Actuel,30), 12],
	Cons_Para_13:= 				Tab_Recette_Auto[0, LIMIT(1,Numero_Etape_Actuel,30), 13],
	Cons_Para_14:= 				Tab_Recette_Auto[0, LIMIT(1,Numero_Etape_Actuel,30), 14],
	Cons_Para_15:= 				Tab_Recette_Auto[0, LIMIT(1,Numero_Etape_Actuel,30), 15],);

(*Lecture des consignes actuel en cours de fonctionnement pour chaque étape (Valeurs en entrées du bloc Mode)*)
Numero_Mode_Actuel 				:= (Mode_Auto.Numero_Mode);
Tempo_Transition_seconde_Actuel := (Mode_Auto.Tempo_Transition_seconde);
Tempo_Transition_Minute_Actuel 	:= (Mode_Auto.Tempo_Transition_Minute);
Tempo_Transition_Heure_Actuel 	:= (Mode_Auto.Tempo_Transition_Heure);
Cons_Volume_Eau_Douche_Actuel 	:= (Mode_Auto.Cons_Volume_Eau_Douche);
Cons_Volume_Eau_Lavabo_Actuel	:= (Mode_Auto.Cons_Volume_Eau_Lavabo);
Cons_Deb_Soufflage_Actuel 		:= (Mode_Auto.Cons_Deb_Soufflage);
Cons_Deb_Extraction_Actuel 		:= (Mode_Auto.Cons_Deb_Extraction);
Cons_Temperature_Eau_Actuel 	:= (Mode_Auto.Cons_Temperature_Eau);
Cons_Para_Nbre_Chasse_Eau 		:= (Mode_Auto.Cons_Nbre_Chasse);
Cons_Para_11_Actuel 			:= (Mode_Auto.Cons_Para_11);
Cons_Para_12_Actuel 			:= (Mode_Auto.Cons_Para_12);
Cons_Para_13_Actuel 			:= (Mode_Auto.Cons_Para_13);
Cons_Para_14_Actuel 			:= (Mode_Auto.Cons_Para_14);
Cons_Para_15_Actuel 			:= (Mode_Auto.Cons_Para_15);

(*Lecture des consignes appliquée en cours de fonctionnement pour chaque étape (Valeurs en sorties du bloc Mode)*)
(*Affichage du texte du mode en cours*)
MEMSET(ADR(Lecture_Texte_Choisi_FR),0,SIZEOF(Lecture_Texte_Choisi_FR));
MEMSET(ADR(Lecture_Texte_Choisi_ENG),0,SIZEOF(Lecture_Texte_Choisi_ENG));
Lecture_Texte_Choisi_FR 	:= Mode_Auto.Out_Texte_FR;
Lecture_Texte_Choisi_ENG	:= Mode_Auto.Out_Texte_ENG;
(*Gestion du décompte du temps restant*)
Temp_Restant_Seconde 			:= Mode_Auto.Out_Restant_Seconde;
Temp_Restant_Minute 			:= Mode_Auto.Out_Restant_Minute;
Temp_Restant_Heure 				:= Mode_Auto.Out_Restant_Heure;
(*Gestion du décompte du nombre de chasse*)
Nbre_Chasse_Total := Mode_Auto.Cons_Nbre_Chasse;
Nbre_Chasse_EnCours := MAX(Mode_Auto.Cpt_Chasse_PV, Mode_Auto.Cpt_Chasse_GV);
(*Débit d'eau, consigne de ventilation et consigne de température d'eau*)
IF (S_Cmd_Vanne_Alim_Douche OR S_Cmd_ElectroValve_Alim_Douche) THEN
Lect_Volume_Eau_Douche 			:= LIMIT(0,(Mode_Auto.Out_Volume_Eau_Douche - Trop_Plein_Douche + Garde_Deau_Douche),150);
ELSE Lect_Volume_Eau_Douche := 0.0; END_IF;
IF (S_Cmd_Vanne_Alim_Lavabo OR S_Cmd_ElectroValve_Alim_Lavabo) THEN
Lect_Volume_Eau_Lavabo			:= LIMIT(0,(Mode_Auto.Out_Volume_Eau_Lavabo - Trop_Plein_Lavabo + Garde_Deau_Lavabo),150);
ELSE Lect_Volume_Eau_Lavabo := 0.0; END_IF;
Cons_Deb_Soufflage_Appli 		:= Mode_Auto.Out_Debit_Souf;
Cons_Deb_Extraction_Appli 		:= Mode_Auto.Out_Debit_Ext;
Cons_Temperature_Eau_Appli 		:= Mode_Auto.Out_Temp_Eau;
Cons_Para_Nbre_Chasse_Eau 		:= Mode_Auto.Cons_Nbre_Chasse;
Cons_Para_11_Appli 				:= Mode_Auto.Out_Para_11;
Cons_Para_12_Appli 				:= Mode_Auto.Out_Para_12;
Cons_Para_13_Appli 				:= Mode_Auto.Out_Para_13;
Cons_Para_14_Appli 				:= Mode_Auto.Out_Para_14;
Cons_Para_15_Appli 				:= Mode_Auto.Out_Para_15;

(*Passage à l'étape suivante*)
R_TRIG1(CLK:= Mode_Auto.Fin_Action);
IF(R_TRIG1.Q)
	THEN
	Numero_Etape_Actuel := Numero_Etape_Actuel + 1;
END_IF;

(*Fin de la recette*)
IF(Mode_Arret_Auto)
	THEN
	Numero_Mode_Auto := 3;
END_IF;

(*******************************************************************************************Gestion vérification de la poste de ventilation*)
3:
(*Attente de quelques secondes si demmande de post ventilation*)
TON_PV(IN:= (NOT Dmd_Post_Ventilation), PT:= T#1s);
R_TRIG_PV(CLK:= TON_PV.Q);
 (*Démarrage de la recette à la fin de la post ventilation*)
F_TRIG_Fin_Post_Ventil(CLK:= Dmd_Post_Ventilation);
IF(F_TRIG_Fin_Post_Ventil.Q OR R_TRIG_PV.Q)
	THEN
	Numero_Mode_Auto := 2;
END_IF;
MEMSET(ADR(Lecture_Texte_Choisi_FR),0,SIZEOF(Lecture_Texte_Choisi_FR));
MEMSET(ADR(Lecture_Texte_Choisi_ENG),0,SIZEOF(Lecture_Texte_Choisi_ENG));
IF (Dmd_Post_Ventilation) (*Affichage du texte post ventilation*)
	THEN
	Lecture_Texte_Choisi_FR 	:= 'POST VENTILATION EN COURS';
	Lecture_Texte_Choisi_ENG	:= 'POST VENTILATION IN PROCESS';
END_IF;
Mode_Auto(
	Enable:= 					FALSE,
	Numero_Etape:= 				0,
	Numero_Mode:= 				0,
	Tempo_Transition_seconde:=	0,
	Tempo_Transition_Minute:=	0,
	Tempo_Transition_Heure:= 	0,
	Cons_Volume_Eau_Douche:= 	0,
	Cons_Volume_Eau_Lavabo:=	0,
	Cons_Deb_Soufflage:= 		0,
	Cons_Deb_Extraction:=		0,
	Cons_Temperature_Eau:= 		0,
	Cons_Nbre_Chasse:= 			0,
	Cons_Para_11:= 				0,
	Cons_Para_12:= 				0,
	Cons_Para_13:= 				0,
	Cons_Para_14:= 				0,
	Cons_Para_15:= 				0);

(*******************************************************************************************Etape 2 : Initialisation des valeurs*)
2:
FOR j := 1 TO 29 BY 1 DO
	Tab_Recette_Auto[0, j, 1] := 0;
	Tab_Recette_Auto[0, j, 2] := 0;
	Tab_Recette_Auto[0, j, 3] := 0;
	Tab_Recette_Auto[0, j, 4] := 0;
	Tab_Recette_Auto[0, j, 5] := 0;
	Tab_Recette_Auto[0, j, 6] := 0;
	Tab_Recette_Auto[0, j, 7] := 0;
	Tab_Recette_Auto[0, j, 8] := 0;
	Tab_Recette_Auto[0, j, 9] := 0;
	Tab_Recette_Auto[0, j, 10] := 0;
	Tab_Recette_Auto[0, j, 11] := 0;
	Tab_Recette_Auto[0, j, 12] := 0;
	Tab_Recette_Auto[0, j, 13] := 0;
	Tab_Recette_Auto[0, j, 14] := 0;
	Tab_Recette_Auto[0, j, 15] := 0;

	Tab_Enr_Recette[0, j, 1] := 0;
	Tab_Enr_Recette[0, j, 2] := 0;
	Tab_Enr_Recette[0, j, 3] := 0;
	Tab_Enr_Recette[0, j, 4] := 0;
	Tab_Enr_Recette[0, j, 5] := 0;
	Tab_Enr_Recette[0, j, 6] := 0;
	Tab_Enr_Recette[0, j, 7] := 0;
	Tab_Enr_Recette[0, j, 8] := 0;
	Tab_Enr_Recette[0, j, 9] := 0;
	Tab_Enr_Recette[0, j, 10] := 0;
	Tab_Enr_Recette[0, j, 11] := 0;
	Tab_Enr_Recette[0, j, 12] := 0;
	Tab_Enr_Recette[0, j, 13] := 0;
	Tab_Enr_Recette[0, j, 14] := 0;
	Tab_Enr_Recette[0, j, 15] := 0;
END_FOR;

Numero_Etape_Actuel := 0;
Nbre_Etape_Totale := 0;

R_TRIG_Dem(CLK:=FALSE);
R_TRIG1(CLK:=FALSE);
F_TRIG_Fin_Post_Ventil(CLK:= FALSE);
TON_PV(IN:= (FALSE));
R_TRIG_PV(CLK:= FALSE);

Numero_Mode_Actuel 				:= 0;
Tempo_Transition_seconde_Actuel := 0;
Tempo_Transition_Minute_Actuel 	:= 0;
Tempo_Transition_Heure_Actuel 	:= 0;
Cons_Volume_Eau_Douche_Actuel 	:= 0;
Cons_Volume_Eau_Lavabo_Actuel	:= 0;
Cons_Deb_Soufflage_Actuel 		:= 0;
Cons_Deb_Extraction_Actuel 		:= 0;
Cons_Temperature_Eau_Actuel 	:= 0;
Cons_Para_Nbre_Chasse_Eau 		:= 0;
Cons_Para_11_Actuel 			:= 0;
Cons_Para_12_Actuel 			:= 0;
Cons_Para_13_Actuel 			:= 0;
Cons_Para_14_Actuel 			:= 0;
Cons_Para_15_Actuel 			:= 0;

Mode_Auto(
	Enable:= 					FALSE,
	Numero_Etape:= 				0,
	Numero_Mode:= 				0,
	Tempo_Transition_seconde:=	0,
	Tempo_Transition_Minute:=	0,
	Tempo_Transition_Heure:= 	0,
	Cons_Volume_Eau_Douche:= 	0,
	Cons_Volume_Eau_Lavabo:=	0,
	Cons_Deb_Soufflage:= 		0,
	Cons_Deb_Extraction:=		0,
	Cons_Temperature_Eau:= 		0,
	Cons_Nbre_Chasse:= 			0,
	Cons_Para_11:= 				0,
	Cons_Para_12:= 				0,
	Cons_Para_13:= 				0,
	Cons_Para_14:= 				0,
	Cons_Para_15:= 				0);

Cons_Dimmer_Auto				:= 254;
Cons_Appl_Rouge_Auto			:= 254;
Cons_Appl_Vert_Auto				:= 254;
Cons_Appl_Bleu_Auto				:= 254;
Cons_Appl_Blanc_Auto			:= 254;

MEMSET(ADR(Lecture_Texte_Choisi_FR),0,SIZEOF(Lecture_Texte_Choisi_FR));
MEMSET(ADR(Lecture_Texte_Choisi_ENG),0,SIZEOF(Lecture_Texte_Choisi_ENG));

Lecture_Texte_Choisi_FR			:= '';
Lecture_Texte_Choisi_ENG		:= '';
Temp_Restant_Seconde 			:= 0.0;
Temp_Restant_Minute 			:= 0.0;
Temp_Restant_Heure 				:= 0.0;
Lect_Volume_Eau_Douche 			:= 0.0;
Lect_Volume_Eau_Lavabo			:= 0.0;
Cons_Deb_Soufflage_Appli 		:= 0.0;
Cons_Deb_Extraction_Appli 		:= 0.0;
Cons_Temperature_Eau_Appli 		:= 0.0;
Cons_Para_Nbre_Chasse_Eau 		:= 0.0;
Cons_Para_11_Appli 				:= 0.0;
Cons_Para_12_Appli 				:= 0.0;
Cons_Para_13_Appli 				:= 0.0;
Cons_Para_14_Appli 				:= 0.0;
Cons_Para_15_Appli 				:= 0.0;

(*Retour à l'étape 0 à la fin de l'initialisation*)
Numero_Mode_Auto := 0;
END_CASE;

END_PROGRAM

// ---- POUs/j_Protocol_Manu.TcPOU
PROGRAM j_Protocol_Manu
VAR
(*Enregistrement de la recette manuel*)
	R_TRIG_Enr_Manuel: R_TRIG;
(*initialisation des valeurs*)
END_VAR

(************************************************************************************************************************Gestion Arrêt du grafcet*)
Mode_Arret_Manu := 	(Reset_Mode_Manu(*Bouton arrêt*)
					OR ((Numero_Mode_Manu = 1) AND Mode_Manu.Fin_Action) (*Fin du mode*)
					OR (Mode_Manu.Mode_12 AND Defaut_Discord_Deb_Eau_Douche)
					OR (Mode_Manu.Mode_13 AND Defaut_Discord_Deb_Eau_Douche)
					OR (Mode_Manu.Mode_14 AND Defaut_Discord_Deb_Eau_Lavabo)
					OR (Mode_Manu.Mode_15 AND Defaut_Discord_Deb_Eau_Lavabo)
					OR Defaut_Debordement_Douche OR Defaut_Debordement_Lavabo)
					OR (Mode_Manu.Mode_4 AND Defaut_Discord_Deb_Eau_Lavabo AND Option_Debitmetre_Lavabo)
					OR (Mode_Manu.Mode_5 AND Defaut_Discord_Deb_Eau_Lavabo AND Option_Debitmetre_Lavabo)
					OR (Mode_Manu.Mode_1 AND Defaut_Discord_Deb_Eau_Douche AND Option_Debitmetre_Douche)
					OR (Mode_Manu.Mode_2 AND Defaut_Discord_Deb_Eau_Douche AND Option_Debitmetre_Douche)
					OR (Mode_Auto.Mode_25 AND Defaut_Arret_Mode25 AND Option_Cabine_Climatique)
					OR Defaut_Discord_Reg_Etanche_Ext OR Defaut_Sonde_Temp_Eau_Mitig;

(************************************************************************************************************************Enregistrement de la recette manuel*)
R_TRIG_Enr_Manuel(CLK:=Mode_Cabine_Manuel);
IF(R_TRIG_Enr_Manuel.Q)
	THEN
	Tab_Enr_Mode_Manu[1] 			:= Manu_Choix_Numero_Mode;
	Tab_Enr_Mode_Manu[2] 			:= Manu_Tempo_Transition_Seconde;
	Tab_Enr_Mode_Manu[3] 			:= Manu_Tempo_Transition_Minute;
	Tab_Enr_Mode_Manu[4] 			:= Manu_Tempo_Transition_Heure;
	Tab_Enr_Mode_Manu[5] 			:= Manu_Lct_Cons_Vol_Douche;
	Tab_Enr_Mode_Manu[6] 			:= Manu_Lct_Cons_Vol_Lavabo;
	Tab_Enr_Mode_Manu[7] 			:= Manu_Cons_Deb_Soufflage;
	Tab_Enr_Mode_Manu[8] 			:= Manu_Cons_Deb_Extraction;
	Tab_Enr_Mode_Manu[9] 			:= Manu_Cons_Temp_Eau;
	Tab_Enr_Mode_Manu[10] 			:= Manu_Cons_Nbre_Chasse;
	Tab_Enr_Mode_Manu[11] 			:= Manu_Cons_Para11;
	Tab_Enr_Mode_Manu[12] 			:= Manu_Cons_Para12;
	Tab_Enr_Mode_Manu[13] 			:= Manu_Cons_Para13;
	Tab_Enr_Mode_Manu[14] 			:= Manu_Cons_Para14;
	Tab_Enr_Mode_Manu[15] 			:= Manu_Cons_Para15;
END_IF;

(************************************************************************************************************************Démarrage du mode manu*)
(*Démarrage du mode manuel à la fin de l'enregistrement*)
IF(Mode_Cabine_Manuel AND (Tab_Enr_Mode_Manu[1] <> 0))
	THEN
	Numero_Mode_Manu := 1;
END_IF;

(*Gestion du case du mode auto*)
CASE Numero_Mode_Manu OF
(*******************************************************************************************Etape 0 : Attente*)
0:
Mode_Manu(
	Enable:= 						(FALSE),
	Numero_Etape:= 					Numero_Mode_Manu);

(*******************************************************************************************Etape 1 : Execution de la recette en mode auto*)
1:
Mode_Manu(
	Enable:= 						(Numero_Mode_Manu = 1),
	Numero_Etape:= 					Numero_Mode_Manu,
	Numero_Mode:= 					Tab_Enr_Mode_Manu[1],
	Tempo_Transition_seconde:= 		Tab_Enr_Mode_Manu[2],
	Tempo_Transition_Minute:=		Tab_Enr_Mode_Manu[3],
	Tempo_Transition_Heure:= 		Tab_Enr_Mode_Manu[4],
	Cons_Volume_Eau_Douche:= 		Tab_Enr_Mode_Manu[5],
	Cons_Volume_Eau_Lavabo:=		Tab_Enr_Mode_Manu[6],
	Cons_Deb_Soufflage:=			Tab_Enr_Mode_Manu[7],
	Cons_Deb_Extraction:=			Tab_Enr_Mode_Manu[8],
	Cons_Temperature_Eau:=			Tab_Enr_Mode_Manu[9],
	Cons_Nbre_Chasse:=				Tab_Enr_Mode_Manu[10],
	Cons_Para_11:=					Tab_Enr_Mode_Manu[11],
	Cons_Para_12:= 					Tab_Enr_Mode_Manu[12],
	Cons_Para_13:=					Tab_Enr_Mode_Manu[13],
	Cons_Para_14:=					Tab_Enr_Mode_Manu[14],
	Cons_Para_15:= 					Tab_Enr_Mode_Manu[15]);

(*Lecture des consignes appliquée en cours de fonctionnement pour chaque étape (Valeurs en sorties du bloc Mode)*)
(*Affichage du texte du mode en cours*)
MEMSET(ADR(Lecture_Texte_Choisi_FR),0,SIZEOF(Lecture_Texte_Choisi_FR));
MEMSET(ADR(Lecture_Texte_Choisi_ENG),0,SIZEOF(Lecture_Texte_Choisi_ENG));
Lecture_Texte_Choisi_FR 			:= Mode_Manu.Out_Texte_FR;
Lecture_Texte_Choisi_ENG			:= Mode_Manu.Out_Texte_ENG;
(*Gestion du décompte du temps restant*)
Temp_Restant_Seconde 				:= Mode_Manu.Out_Restant_Seconde;
Temp_Restant_Minute 				:= Mode_Manu.Out_Restant_Minute;
Temp_Restant_Heure 					:= Mode_Manu.Out_Restant_Heure;
(*Gestion du décompte du nombre de chasse*)
Nbre_Chasse_Total 					:= Mode_Manu.Cons_Nbre_Chasse;
Nbre_Chasse_EnCours 				:= MAX(Mode_Manu.Cpt_Chasse_PV, Mode_Manu.Cpt_Chasse_GV);
(*Débit d'eau, consigne de ventilation et consigne de température d'eau*)
IF (S_Cmd_Vanne_Alim_Douche OR S_Cmd_ElectroValve_Alim_Douche) THEN
Lect_Volume_Eau_Douche 				:= LIMIT(0,(Mode_Manu.Out_Volume_Eau_Douche - Trop_Plein_Douche + Garde_Deau_Douche),150);
ELSE Lect_Volume_Eau_Douche 		:= 0.0; END_IF;
IF (S_Cmd_Vanne_Alim_Lavabo OR S_Cmd_ElectroValve_Alim_Lavabo) THEN
Lect_Volume_Eau_Lavabo				:= LIMIT(0,(Mode_Manu.Out_Volume_Eau_Lavabo - Trop_Plein_Lavabo + Garde_Deau_Lavabo),150);
ELSE Lect_Volume_Eau_Lavabo 		:= 0.0; END_IF;
Cons_Deb_Soufflage_Appli 			:= Mode_Manu.Out_Debit_Souf;
Cons_Deb_Extraction_Appli 			:= Mode_Manu.Out_Debit_Ext;
Cons_Temperature_Eau_Appli 			:= Mode_Manu.Out_Temp_Eau;
Cons_Para_Nbre_Chasse_Eau 			:= Mode_Manu.Cons_Nbre_Chasse;
Cons_Para_11_Appli 					:= Mode_Manu.Out_Para_11;
Cons_Para_12_Appli 					:= Mode_Manu.Out_Para_12;
Cons_Para_13_Appli 					:= Mode_Manu.Out_Para_13;
Cons_Para_14_Appli 					:= Mode_Manu.Out_Para_14;
Cons_Para_15_Appli 					:= Mode_Manu.Out_Para_15;

(*Fin du mode*)
IF(Mode_Arret_Manu)
	THEN
	Numero_Mode_Manu := 2;
END_IF;

(*******************************************************************************************Etape 2 : Initialisation des valeurs*)
2:
Tab_Enr_Mode_Manu[1] 				:= 0;
Tab_Enr_Mode_Manu[2] 				:= 0;
Tab_Enr_Mode_Manu[3] 				:= 0;
Tab_Enr_Mode_Manu[4] 				:= 0;
Tab_Enr_Mode_Manu[5] 				:= 0;
Tab_Enr_Mode_Manu[6] 				:= 0;
Tab_Enr_Mode_Manu[7] 				:= 0;
Tab_Enr_Mode_Manu[8] 				:= 0;
Tab_Enr_Mode_Manu[9] 				:= 0;
Tab_Enr_Mode_Manu[10]				:= 0;
Tab_Enr_Mode_Manu[11]				:= 0;
Tab_Enr_Mode_Manu[12]				:= 0;
Tab_Enr_Mode_Manu[13]				:= 0;
Tab_Enr_Mode_Manu[14]				:= 0;
Tab_Enr_Mode_Manu[15]				:= 0;

Mode_Manu(
	Enable:= 						FALSE,
	Numero_Etape:= 					0,
	Numero_Mode:= 					0,
	Tempo_Transition_seconde:=		0,
	Tempo_Transition_Minute:=		0,
	Tempo_Transition_Heure:= 		0,
	Cons_Volume_Eau_Douche:= 		0,
	Cons_Volume_Eau_Lavabo:=		0,
	Cons_Deb_Soufflage:= 			0,
	Cons_Deb_Extraction:=			0,
	Cons_Temperature_Eau:= 			0,
	Cons_Nbre_Chasse:= 				0,
	Cons_Para_11:= 					0,
	Cons_Para_12:= 					0,
	Cons_Para_13:= 					0,
	Cons_Para_14:= 					0,
	Cons_Para_15:= 					0);

MEMSET(ADR(Lecture_Texte_Choisi_FR),0,SIZEOF(Lecture_Texte_Choisi_FR));
MEMSET(ADR(Lecture_Texte_Choisi_ENG),0,SIZEOF(Lecture_Texte_Choisi_ENG));
Lecture_Texte_Choisi_FR				:= '';
Lecture_Texte_Choisi_ENG			:= '';
Temp_Restant_Seconde 				:= 0.0;
Temp_Restant_Minute 				:= 0.0;
Temp_Restant_Heure 					:= 0.0;
Lect_Volume_Eau_Douche 				:= 0.0;
Lect_Volume_Eau_Lavabo				:= 0.0;
Cons_Deb_Soufflage_Appli 			:= 0.0;
Cons_Deb_Extraction_Appli 			:= 0.0;
Cons_Temperature_Eau_Appli 			:= 0.0;
Cons_Para_Nbre_Chasse_Eau 			:= 0.0;
Cons_Para_11_Appli 					:= 0.0;
Cons_Para_12_Appli 					:= 0.0;
Cons_Para_13_Appli 					:= 0.0;
Cons_Para_14_Appli 					:= 0.0;
Cons_Para_15_Appli 					:= 0.0;

(*Retour à l'étape 0 à la fin de l'initialisation*)
Numero_Mode_Manu 					:= 0;
END_CASE;

END_PROGRAM

// ---- POUs/l_Cons_LED.TcPOU
PROGRAM l_Cons_LED
VAR
	Pulse_Defaut_Led_Cabine:BOOL;
	BLINK_Defaut: BLINK;
END_VAR

(*********************************Gestion du clignotement lors d'un défaut**********************************)
BLINK_Defaut(ENABLE:= (Mode_Cabine_Defaut), TIMELOW:= T#2s, TIMEHIGH:= T#2s, OUT=> Pulse_Defaut_Led_Cabine);

(******************************************Mode Maintenance (orange)*****************************************)
IF(Mode_Maintenance)
	THEN
	Cde_Dimmer_Cabine		:= 254;
	Cde_Rouge_Cabine		:= 254;
	Cde_Vert_Cabine			:= 127;
	Cde_Bleu_Cabine			:= 0;
	Cde_Blanc_Cabine		:= 0;
END_IF;

(*******************************************Mode cabine libre (Vert)********************************************)
IF(Mode_Cabine_Libre)
	THEN
	Cde_Dimmer_Cabine		:= 254;
	Cde_Rouge_Cabine		:= WORD_TO_INT(Cde_Rouge_Cabine_Libre);
	Cde_Vert_Cabine			:= WORD_TO_INT(Cde_Vert_Cabine_Libre);
	Cde_Bleu_Cabine			:= WORD_TO_INT(Cde_Bleu_Cabine_Libre);
	Cde_Blanc_Cabine		:= WORD_TO_INT(Cde_Blanc_Cabine_Libre);
END_IF;

(*****************************************Mode cabine manuel (Bleu)******************************************)
IF(Mode_Cabine_Manuel)
	THEN
	Cde_Dimmer_Cabine		:= 254;
	Cde_Rouge_Cabine		:= 0;
	Cde_Vert_Cabine			:= 0;
	Cde_Bleu_Cabine			:= 254;
	Cde_Blanc_Cabine		:= 0;
END_IF;

(***************************Mode cabine automatique (Utilisateur)***************************)
IF(Mode_Cabine_Automatique)
	THEN
	Cde_Dimmer_Cabine		:= Cons_Dimmer_Auto;
	Cde_Rouge_Cabine		:= Cons_Appl_Rouge_Auto;
	Cde_Vert_Cabine			:= Cons_Appl_Vert_Auto;
	Cde_Bleu_Cabine			:= Cons_Appl_Bleu_Auto;
	Cde_Blanc_Cabine		:= Cons_Appl_Blanc_Auto;
END_IF;

(**************************************Mode cabine dépollution (Rouge)***************************************)
IF(Mode_Cabine_Depollution)
	THEN
	Cde_Dimmer_Cabine		:= 254;
	Cde_Rouge_Cabine		:= 254;
	Cde_Vert_Cabine			:= 0;
	Cde_Bleu_Cabine			:= 0;
	Cde_Blanc_Cabine		:= 0;
END_IF;

(**************************************Mode cabine en défaut (rouge clignotant)*******************************)
IF(Mode_Cabine_Defaut AND Pulse_Defaut_Led_Cabine)
	THEN
	Cde_Dimmer_Cabine		:= 254;
	Cde_Rouge_Cabine		:= 254;
	Cde_Vert_Cabine			:= 0;
	Cde_Bleu_Cabine			:= 0;
	Cde_Blanc_Cabine		:= 0;
END_IF;
IF(Mode_Cabine_Defaut AND NOT Pulse_Defaut_Led_Cabine)
	THEN
	Cde_Dimmer_Cabine		:= 0;
	Cde_Rouge_Cabine		:= 0;
	Cde_Vert_Cabine			:= 0;
	Cde_Bleu_Cabine			:= 0;
	Cde_Blanc_Cabine		:= 0;
END_IF;

(*************************************************Mode éclairage (blanc)******************************************)
IF(Mode_Cabine_Eclairage OR Mode_Cabine_Nettoyage)
	THEN
	Cde_Dimmer_Cabine		:= 254;
	Cde_Rouge_Cabine		:= 254;
	Cde_Vert_Cabine			:= 254;
	Cde_Bleu_Cabine			:= 254;
	Cde_Blanc_Cabine		:= 254;
END_IF;

END_PROGRAM

// ---- POUs/n0_Regulation_Bas_Deb.TcPOU
PROGRAM n0_Regulation_Bas_Deb
VAR
	PID_Bas_Deb_Ext: PID;
	Var_Interne: REAL;
END_VAR

(**********************************************Gestion de l'enable de la régulation PID*)
(*Vérification que la conisgne appliquée est compris dans la consigne bas débit*)
IF((Cons_Actionneur_Registre_Souf_Volh > 0) AND (Cons_Actionneur_Registre_Souf_Volh <= Cons_Max_Bas_Deb_Ext) AND Option_Bas_Debit)
	THEN
	IF (E_Vanne_Souf_Bas_Deb_Ouv AND E_Vanne_Ext_Bas_Deb_Ouv)
		THEN
		Enable_PID_Bas_Deb_Ext := TRUE;
		ELSE
		Enable_PID_Bas_Deb_Ext := FALSE;
	END_IF;
	Cmd_Appli_Vanne_Souf_Bas_Deb := TRUE;
	Cmd_Appli_Vanne_Ext_Bas_Deb := TRUE;
	ELSE
	Enable_PID_Bas_Deb_Ext := FALSE;
	Cmd_Appli_Vanne_Souf_Bas_Deb := FALSE;
	Cmd_Appli_Vanne_Ext_Bas_Deb := FALSE;
END_IF;

Var_Interne := LIMIT(0.0,Cons_Actionneur_Registre_Souf_m3h, 16.0);

(**********************************************Régulation PID*)
PID_Bas_Deb_Ext(
	ACTUAL:= MES_Petit_Debit_m3h_Extraction,
	SET_POINT:= Var_Interne, (*Recopie de la consigne de soufflage pour la consigne du bas débit*)
	KP:= Gain_PID_Bas_Deb_Ext,
	TN:= Integral_PID_Bas_Deb_Ext,
	TV:= Derivee_PID_Bas_Deb_Ext,
	Y_MANUAL:= 0.0,
	Y_OFFSET:= 0.0,
	Y_MIN:= 0.0,
	Y_MAX:= 100.0,
	RESET:= NOT Enable_PID_Bas_Deb_Ext, (* Attente ouvertures des registres avant de démarrer la régulation*)
	Y=> S_Cmd_PID_Bas_Deb_Ext);

(*Consigne actionneur*)
Cons_Actionneur_Moteur_BasDebit := S_Cmd_PID_Bas_Deb_Ext;

END_PROGRAM

// ---- POUs/n1_Regulation_Press.TcPOU
PROGRAM n1_Regulation_Press
VAR
	TON_1 :TON;
	PID_Press: PID;
	Valeur_Trunc_Press: REAL;
	Gain_Negatif: REAL;
	Enable_PID_Press :BOOL;
	TOF_1: TOF;
END_VAR

(**********************************************Gestion de l'enable de la régulation PID*)
(*Gestion de la régulation de la pression uniquement si consigne supérieur à au minimum du bas débit*)
TON_1(IN:= ((Cons_Actionneur_Registre_Ext_m3h > ((Cons_Max_Bas_Deb_Ext + 0.5) * Volume_Cabine))) AND Option_Regul_Deb_Ou_Press, PT:= T#2s);
IF((TON_1.Q AND NOT Mode_Auto.Mode_25) OR Dmd_Post_Ventilation)
	THEN
	Enable_PID_Press := TRUE;
	ELSE
	Enable_PID_Press := FALSE;
END_IF;

(*Gestion d'un TOF afin d'éviter de fermer trop rapidement le registre car le registre soufflage est plus lent*)
TOF_1(IN:= Enable_PID_Press, PT:= T#30s);
Enable_PID_Press_Cab := TOF_1.Q;

Valeur_Trunc_Press := DINT_TO_REAL(TRUNC(Tab_MES_Sonde_Press_Cab.R_MesCor));
Gain_Negatif := Gain_PID_Press_Cab *  -1.0;

(**********************************************Régulation PID*)
PID_Press(
	ACTUAL:= Valeur_Trunc_Press,
	SET_POINT:= Cons_Press_Cab,
	KP:= Gain_Negatif,
	TN:= Integral_PID_Press_Cab,
	TV:= Derivee_PID_Press_Cab,
	Y_MANUAL:= 0.0,
	Y_OFFSET:= 0.0,
	Y_MIN:= 0.0,
	Y_MAX:= 100.0,
	RESET:= NOT Enable_PID_Press_Cab,
	Y=> S_Cmd_PID_Press_Cab);

S_Ecart_Regul_PID_Pression := SEL(Enable_PID_Press_Cab, 0.0, ABS(PID_Press.ERROR));

END_PROGRAM

// ---- POUs/n2_Regulation_Temp.TcPOU
PROGRAM n2_Regulation_Temp
VAR
	TON_1: TON;
	TON_2: TON;
	PID_Temp: PID;
END_VAR

(**********************************************Gestion de l'enable de la régulation PID*)
(*Gestion de la régulation de la batterie uniquement s'il n'y a pas de défaut et s'il y ' a présence d'un débit de soufflage*)
TON_1(IN:= (Tab_MES_Sonde_Gros_Debit_Soufflage.R_MesCor > 50.0), PT:= T#1m);
IF(NOT Defaut_Klixon_BattElec AND TON_1.Q AND Option_Batt_Elec)
	THEN
	Enable_PID_Temp_Amb := TRUE;
	ELSE
	Enable_PID_Temp_Amb := FALSE;
END_IF;

(**********************************************Régulation PID*)
PID_Temp(
	ACTUAL:= Tab_MES_Sonde_Temp_Amb.R_MesCor,
	SET_POINT:= Cons_Temp_Amb,
	KP:= Gain_PID_Temp_Amb,
	TN:= Integral_PID_Temp_Amb,
	TV:= Derivee_PID_Temp_Amb,
	Y_MANUAL:= 0.0,
	Y_OFFSET:= 0.0,
	Y_MIN:= 0.0,
	Y_MAX:= 100.0,
	RESET:= NOT Enable_PID_Temp_Amb,
	Y=> S_Cmd_PID_Temp_Amb);

Cons_Actionneur_BattElec := S_Cmd_PID_Temp_Amb;
(*Gestion de la commande du contacteur si demande PID supérieure à 5%*)
TON_2(IN:= (S_Cmd_PID_Temp_Amb > 5.0), PT:= T#1m);
IF(TON_2.Q AND Enable_PID_Temp_Amb)
	THEN
	Cmd_Appli_BattElec := TRUE;
	ELSE
	Cmd_Appli_BattElec := FALSE;
END_IF;

END_PROGRAM

// ---- POUs/n3_Regul_Temp_EauMitig.TcPOU
PROGRAM n3_Regul_Temp_EauMitig
VAR
	PID_Temp_Eau_Mitig: PID;
	SetPoint_PID_Temp_EM: REAL;
	Actual_PID_Temp_EM: REAL;
	TON_1: TON;
END_VAR

(**********************************************Gestion de l'enable de la régulation PID*)
(*Gestion de la régulation de la température uniquement si une d'alimentation est ouverte (sauf NEP et douchette)*)
(*Petite temporisation le temps que la température bouge après une ouverture de vanne*)
TON_1(IN:= ((E_Vanne_Alim_Douche_Ouv OR E_Vanne_Alim_Lavabo_Ouv OR S_Cmd_ElectroValve_Alim_Douche OR S_Cmd_ElectroValve_Alim_Lavabo) AND Option_Regul_Temp_Eau), PT:= T#5S);
IF (TON_1.Q)
	THEN
	Enable_PID_Temp_Eau_Mitig := TRUE;
	ELSE
	Enable_PID_Temp_Eau_Mitig := FALSE;
END_IF;

(*Gestion de la consigne celon le mode*)
IF (Mode_Cabine_Automatique) THEN (*SetPoint_PID_Temp_EM := Mode_Auto.Out_Temp_Eau*) SetPoint_PID_Temp_EM := Cons_Temp_EauMitige ; END_IF;
IF (Mode_Cabine_Manuel) THEN SetPoint_PID_Temp_EM := Mode_Manu.Out_Temp_Eau ; END_IF;

(*Gestion du blocage du PID*)
Actual_PID_Temp_EM := SEL(Enable_PID_Temp_Eau_Mitig, SetPoint_PID_Temp_EM ,Tab_MES_Sonde_Temp_Eau_Mitig.R_MesCor);

(**********************************************Régulation PID*)
PID_Temp_Eau_Mitig(
	ACTUAL:= Actual_PID_Temp_EM,
	SET_POINT:= SetPoint_PID_Temp_EM,
	KP:= Gain_PID_Temp_Eau_Mitig,
	TN:= Integral_PID_Temp_Eau_Mitig,
	TV:= Derivee_PID_Temp_Eau_Mitig,
	Y_MANUAL:= 0.0,
	Y_OFFSET:= 0.0,
	Y_MIN:= 0.0,
	Y_MAX:= 100.0,
	RESET:= FALSE,
	Y=> S_Cmd_PID_Temp_Eau_Mitig);

S_Ecart_Regul_PID_Temp_Eau_Mitig := SEL(Enable_PID_Temp_Eau_Mitig, 0.0, ABS(PID_Temp_Eau_Mitig.ERROR));

END_PROGRAM

// ---- POUs/o_Cons_Cmd_Actionneurs.TcPOU
PROGRAM o_Cons_Cmd_Actionneurs
VAR
	Calcul_Temp1: REAL;
	Mode_NEP_Chaud: BOOL;
	Mode_NEP_Froid: BOOL;
	Calcul_Debit_Bypass: REAL;
	ACH_Deb_Souf_Etat_Depol: REAL;
	ACH_Deb_Souf_Etat_Libre: REAL;
	ACH_Mode_Auto_Out_Debit_Souf: REAL;
	Consigne_Mode_EnFctnmnt_PD: REAL := 67.0;
	Consigne_Mode_EnFctnmnt_GD: REAL := 600.0;
END_VAR

(**********************************************Commande des actionneurs*)
Cmd_Appli_PC_Cab					:= (Mode_Auto.Cmd_Prise  AND Mode_Auto.Enable) OR (Mode_Manu.Cmd_Prise AND Mode_Manu.Enable);
Cmd_Appli_Vanne_Alim_Douche			:= (Mode_Auto.Cmd_Douche  AND Mode_Auto.Enable) OR (Mode_Manu.Cmd_Douche AND Mode_Manu.Enable) OR Forc_Ouv_Alim_Lav_Dou;
Cmd_Appli_Vanne_Alim_Douchette		:= ((Mode_Auto.Cmd_Douchette  AND Mode_Auto.Enable) OR (Mode_Manu.Cmd_Douchette AND Mode_Manu.Enable) OR Mode_Cabine_Nettoyage);
Cmd_Appli_Vanne_Alim_Lavabo			:= (Mode_Auto.Cmd_Lavabo  AND Mode_Auto.Enable) OR (Mode_Manu.Cmd_Lavabo AND Mode_Manu.Enable);
Cmd_Appli_Vanne_Vid_Douche			:= ((Mode_Auto.Cmd_Vidange_Douche  AND Mode_Auto.Enable) OR (Mode_Manu.Cmd_Vidange_Douche AND Mode_Manu.Enable) OR Mode_Cabine_Nettoyage);
Cmd_Appli_Vanne_Vid_Lavabo			:= ((Mode_Auto.Cmd_Vidange_Lavabo  AND Mode_Auto.Enable) OR (Mode_Manu.Cmd_Vidange_Lavabo AND Mode_Manu.Enable) OR Mode_Cabine_Nettoyage);
Cmd_Appli_ElectroValve_Alim_Douche	:= (Mode_Auto.Cmd_Electrovanne_Douche  AND Mode_Auto.Enable) OR (Mode_Manu.Cmd_Electrovanne_Douche AND Mode_Manu.Enable);
Cmd_Appli_ElectroValve_Alim_Lavabo	:= (Mode_Auto.Cmd_Electrovanne_Lavabo  AND Mode_Auto.Enable) OR (Mode_Manu.Cmd_Electrovanne_Lavabo AND Mode_Manu.Enable) OR Forc_Ouv_Alim_Lav_Dou;
Cmd_Appli_Reg_Etanche_Souf			:= (Cons_Actionneur_Registre_Souf_m3h > ((Cons_Max_Bas_Deb_Ext + 0.5) * Volume_Cabine)) AND Option_Reg_Etanche_Souf;
Cmd_Appli_Vanne_Alim_NEP			:=  (Mode_Auto.Cmd_NEP  AND Mode_Auto.Enable) OR (Mode_Manu.Cmd_NEP AND Mode_Manu.Enable);
Cmd_Appli_Verin_WC_GV				:=(Mode_Auto.Cmd_Verin_WC_GV  AND Mode_Auto.Enable) OR (Mode_Manu.Cmd_Verin_WC_GV AND Mode_Manu.Enable);
Cmd_Appli_Verin_WC_PV				:=(Mode_Auto.Cmd_Verin_WC_PV  AND Mode_Auto.Enable) OR (Mode_Manu.Cmd_Verin_WC_PV AND Mode_Manu.Enable);

(*Convertion des valeurs m3/h en Vol/h (ACH)*)
ACH_Deb_Souf_Etat_Depol 	:= Cons_Deb_Souf_Etat_Depol * Volume_Cabine;
ACH_Deb_Souf_Etat_Libre 	:= Cons_Deb_Souf_Etat_Libre * Volume_Cabine;
ACH_Mode_Auto_Out_Debit_Souf:= Mode_Auto.Out_Debit_Souf * Volume_Cabine;

(**********************************************Gestion de la consigne de débit en état cabine libre*)
IF(Mode_Cabine_Libre)
	THEN
	Cons_Actionneur_Registre_Ext_Volh 					:= ACH_Deb_Souf_Etat_Libre;
	Cons_Actionneur_Registre_Souf_Volh 					:= ACH_Deb_Souf_Etat_Libre;
	
	IF (ACH_Deb_Souf_Etat_Libre < 354.0) //Mettre la valeur maximum du débit du registre en diam 100mm
		THEN
		GVL_RegTROX.ConsAppliDeb_RegSouf_GD_FCVT01		:= 0.0;
		GVL_RegTROX.ConsAppliDeb_RegSouf_PD_FCVT02		:= ACH_Deb_Souf_Etat_Libre;
		ELSE
		GVL_RegTROX.ConsAppliDeb_RegSouf_GD_FCVT01		:= ACH_Deb_Souf_Etat_Libre;
		GVL_RegTROX.ConsAppliDeb_RegSouf_PD_FCVT02		:= 0.0;	
	END_IF
	GVL_RegTROX.ConsAppliDeb_RegSouf_Cabine_FCVT03		:= 1020.0; //Mettre le débit maximum pour qu'il reste ouvert à 100%
	GVL_RegTROX.ConsAppliDeb_Reg_Bypass_FCVT04			:= 0.0;
	GVL_RegTROX.ConsAppliDeb_RegSouf_CabGD_FCVT05		:= 0.0;
	GVL_RegTROX.ConsAppliDeb_RegSouf_CabPD_FCVT06		:= 0.0;
	GVL_RegTROX.ConsAppliDeb_RegRep_FCVT07				:= 0.0;
END_IF;

(**********************************************Gestion de la consigne de débit en etat cabine dépollution*)
IF(Mode_Cabine_Depollution OR Mode_Depollution_cycle1)
	THEN
	IF (Mode_Depollution_cycle1) // 1er cycle, décontamination de la CTA
		THEN
		Cons_Actionneur_Registre_Ext_Volh 					:= ACH_Deb_Souf_Etat_Depol;
		Cons_Actionneur_Registre_Souf_Volh 					:= ACH_Deb_Souf_Etat_Depol;
		
		GVL_RegTROX.ConsAppliDeb_RegSouf_GD_FCVT01			:= 375.0;
		GVL_RegTROX.ConsAppliDeb_RegSouf_PD_FCVT02			:= 100.0;
		GVL_RegTROX.ConsAppliDeb_RegSouf_Cabine_FCVT03		:= 0.0;
		GVL_RegTROX.ConsAppliDeb_Reg_Bypass_FCVT04			:= 0.0;
		GVL_RegTROX.ConsAppliDeb_RegSouf_CabGD_FCVT05		:= 575.0;
		GVL_RegTROX.ConsAppliDeb_RegSouf_CabPD_FCVT06		:= 100.0;
		GVL_RegTROX.ConsAppliDeb_RegRep_FCVT07				:= 200.0;
	END_IF;
	IF (Mode_Cabine_Depollution AND NOT Mode_Depollution_cycle1) // 2ème cycle, décontamination de la cabine
		THEN
		Cons_Actionneur_Registre_Ext_Volh 					:= ACH_Deb_Souf_Etat_Depol;
		Cons_Actionneur_Registre_Souf_Volh 					:= ACH_Deb_Souf_Etat_Depol;
		
		GVL_RegTROX.ConsAppliDeb_RegSouf_GD_FCVT01			:= ACH_Deb_Souf_Etat_Depol;
		GVL_RegTROX.ConsAppliDeb_RegSouf_PD_FCVT02			:= 0.0;
		GVL_RegTROX.ConsAppliDeb_RegSouf_Cabine_FCVT03		:= 1020.0; //Mettre le débit maximum pour qu'il reste ouvert à 100%
		GVL_RegTROX.ConsAppliDeb_Reg_Bypass_FCVT04			:= 0.0;
		GVL_RegTROX.ConsAppliDeb_RegSouf_CabGD_FCVT05		:= 0.0;
		GVL_RegTROX.ConsAppliDeb_RegSouf_CabPD_FCVT06		:= 0.0;
		GVL_RegTROX.ConsAppliDeb_RegRep_FCVT07				:= 0.0;
	END_IF;
END_IF;

(**********************************************Gestion de la consigne de débit en etat cabine Mode mise en condition*)
IF(Mode_MEnCond AND NOT Mode_Cabine_Libre)
	THEN
	Cons_Actionneur_Registre_Ext_Volh 					:= ACH_Mode_Auto_Out_Debit_Souf;
	Cons_Actionneur_Registre_Souf_Volh 					:= ACH_Mode_Auto_Out_Debit_Souf;
	
	GVL_RegTROX.ConsAppliDeb_RegSouf_GD_FCVT01			:= 0.0;
	GVL_RegTROX.ConsAppliDeb_RegSouf_PD_FCVT02			:= 0.0;
	GVL_RegTROX.ConsAppliDeb_RegSouf_Cabine_FCVT03		:= 0.0;
	GVL_RegTROX.ConsAppliDeb_Reg_Bypass_FCVT04			:= 0.0;
	IF (ACH_Mode_Auto_Out_Debit_Souf < 354.0)  //Mettre la valeur maximum du débit du registre en diam 100mm
		THEN
		GVL_RegTROX.ConsAppliDeb_RegSouf_CabGD_FCVT05	:= 0.0;
		GVL_RegTROX.ConsAppliDeb_RegSouf_CabPD_FCVT06	:= ACH_Mode_Auto_Out_Debit_Souf;
		ELSE
		GVL_RegTROX.ConsAppliDeb_RegSouf_CabGD_FCVT05	:= ACH_Mode_Auto_Out_Debit_Souf;
		GVL_RegTROX.ConsAppliDeb_RegSouf_CabPD_FCVT06	:= 0.0;	
	END_IF
	GVL_RegTROX.ConsAppliDeb_RegRep_FCVT07				:= 1020.0; //Mettre le débit maximum pour qu'il reste ouvert à 100%
END_IF;

(**********************************************Gestion de la consigne de débit en etat cabine Mode fonctionnement*)
IF(Mode_Fctnmt AND NOT Mode_Cabine_Libre)
	THEN
	Cons_Actionneur_Registre_Ext_Volh 					:= ACH_Mode_Auto_Out_Debit_Souf;
	Cons_Actionneur_Registre_Souf_Volh 					:= ACH_Mode_Auto_Out_Debit_Souf;
	(*IF (ACH_Mode_Auto_Out_Debit_Souf < 354.0) //Mettre la valeur maximum du débit du registre en diam 100mm
		THEN
		GVL_RegTROX.ConsAppliDeb_RegSouf_GD_FCVT01		:= 0.0;
		GVL_RegTROX.ConsAppliDeb_RegSouf_PD_FCVT02		:= ACH_Mode_Auto_Out_Debit_Souf;
		ELSE
		GVL_RegTROX.ConsAppliDeb_RegSouf_GD_FCVT01		:= ACH_Mode_Auto_Out_Debit_Souf;
		GVL_RegTROX.ConsAppliDeb_RegSouf_PD_FCVT02		:= 0.0;	
	END_IF*)
	GVL_RegTROX.ConsAppliDeb_RegSouf_GD_FCVT01			:= 0.0;
	GVL_RegTROX.ConsAppliDeb_RegSouf_PD_FCVT02			:= ACH_Mode_Auto_Out_Debit_Souf;
	GVL_RegTROX.ConsAppliDeb_RegSouf_Cabine_FCVT03		:= 0.0;
	Calcul_Debit_Bypass 								:= LIMIT(0.0, 600.0 - (Consigne_Mode_EnFctnmnt_GD + ACH_Mode_Auto_Out_Debit_Souf), 579.0);
	GVL_RegTROX.ConsAppliDeb_Reg_Bypass_FCVT04			:= Calcul_Debit_Bypass;
	GVL_RegTROX.ConsAppliDeb_RegSouf_CabGD_FCVT05		:= Consigne_Mode_EnFctnmnt_GD;
	GVL_RegTROX.ConsAppliDeb_RegSouf_CabPD_FCVT06		:= 0.0;
	(*IF (ACH_Mode_Auto_Out_Debit_Souf < 354.0) //Mettre la valeur maximum du débit du registre en diam 100mm
		THEN
		GVL_RegTROX.ConsAppliDeb_RegSouf_CabGD_FCVT05	:= 0.0;
		GVL_RegTROX.ConsAppliDeb_RegSouf_CabPD_FCVT06	:= ACH_Mode_Auto_Out_Debit_Souf;
		ELSE
		GVL_RegTROX.ConsAppliDeb_RegSouf_CabGD_FCVT05	:= ACH_Mode_Auto_Out_Debit_Souf;
		GVL_RegTROX.ConsAppliDeb_RegSouf_CabPD_FCVT06	:= 0.0;	
	END_IF*)
	GVL_RegTROX.ConsAppliDeb_RegRep_FCVT07				:= LIMIT(0, Consigne_Mode_EnFctnmnt_GD - ACH_Mode_Auto_Out_Debit_Souf, 1020.0);
END_IF;

(**********************************************Consigne des actionneurs en mode manuel*)
IF(Mode_Cabine_Manuel)
	THEN
	Cons_Actionneur_Registre_Ext_Volh 					:= Cons_Deb_Soufflage_Appli;
	Cons_Actionneur_Registre_Souf_Volh 					:= Cons_Deb_Soufflage_Appli;
	IF (Cons_Deb_Soufflage_Appli < 354.0) //Mettre la valeur maximum du débit du registre en diam 100mm
		THEN
		GVL_RegTROX.ConsAppliDeb_RegSouf_GD_FCVT01		:= 0.0;
		GVL_RegTROX.ConsAppliDeb_RegSouf_PD_FCVT02		:= Cons_Deb_Soufflage_Appli;
		ELSE
		GVL_RegTROX.ConsAppliDeb_RegSouf_GD_FCVT01		:= Cons_Deb_Soufflage_Appli;
		GVL_RegTROX.ConsAppliDeb_RegSouf_PD_FCVT02		:= 0.0;	
	END_IF
	GVL_RegTROX.ConsAppliDeb_RegSouf_Cabine_FCVT03		:= 0.0;
	GVL_RegTROX.ConsAppliDeb_Reg_Bypass_FCVT04			:= 0.0;
	GVL_RegTROX.ConsAppliDeb_RegSouf_CabGD_FCVT05		:= 0.0;
	GVL_RegTROX.ConsAppliDeb_RegSouf_CabPD_FCVT06		:= 0.0;
	GVL_RegTROX.ConsAppliDeb_RegRep_FCVT07				:= 0.0;
END_IF;

(**********************************************Gestion des consignes en cas de défaut sur le capteur de pression*)
IF (Defaut_Sonde_Press_Cabine AND NOT Dmd_Post_Ventilation)
	THEN
	GVL_RegTROX.ConsAppliDeb_RegSouf_GD_FCVT01			:= 0.0;
	GVL_RegTROX.ConsAppliDeb_RegSouf_PD_FCVT02			:= 0.0;	
	GVL_RegTROX.ConsAppliDeb_RegSouf_Cabine_FCVT03		:= 0.0;
	GVL_RegTROX.ConsAppliDeb_Reg_Bypass_FCVT04			:= 0.0;
	GVL_RegTROX.ConsAppliDeb_RegSouf_CabGD_FCVT05		:= 0.0;
	GVL_RegTROX.ConsAppliDeb_RegSouf_CabPD_FCVT06		:= 0.0;
	GVL_RegTROX.ConsAppliDeb_RegRep_FCVT07				:= 0.0;
END_IF

(**********************************************Consigne des actionneurs en mode automatique*)
IF(Mode_Cabine_Automatique AND NOT Mode_Cabine_Depollution AND NOT Mode_MEnCond AND NOT Mode_Fctnmt)
	THEN
	Cons_Actionneur_Registre_Ext_Volh	:= Cons_Deb_Soufflage_Appli;
	Cons_Actionneur_Registre_Souf_Volh	:= Cons_Deb_Soufflage_Appli;
	Cons_Actionneur_Moteur_ByPass		:= Mode_Auto.Out_Cons_Moteur_ByPass;
	// Deux types de fonctionnement, la première si une reccette est déclaré avec une gestion de CTA et le deuxième type sans gestion de CTA
	IF (RS_MEnCond.Q1)// gestion avec CTA (Activation des redistres de soufflage générale et du soufflage de la cabine)
		THEN
		Cons_Actionneur_Registre_Ext_Volh 					:= ACH_Mode_Auto_Out_Debit_Souf;
		Cons_Actionneur_Registre_Souf_Volh 					:= ACH_Mode_Auto_Out_Debit_Souf;
		(*IF (ACH_Mode_Auto_Out_Debit_Souf < 354.0) //Mettre la valeur maximum du débit du registre en diam 100mm
			THEN
			GVL_RegTROX.ConsAppliDeb_RegSouf_GD_FCVT01		:= 0.0;
			GVL_RegTROX.ConsAppliDeb_RegSouf_PD_FCVT02		:= ACH_Mode_Auto_Out_Debit_Souf;
			ELSE
			GVL_RegTROX.ConsAppliDeb_RegSouf_GD_FCVT01		:= ACH_Mode_Auto_Out_Debit_Souf;
			GVL_RegTROX.ConsAppliDeb_RegSouf_PD_FCVT02		:= 0.0;	
		END_IF*)
		GVL_RegTROX.ConsAppliDeb_RegSouf_GD_FCVT01			:= 0.0;
		GVL_RegTROX.ConsAppliDeb_RegSouf_PD_FCVT02			:= Consigne_Mode_EnFctnmnt_PD;
		GVL_RegTROX.ConsAppliDeb_RegSouf_Cabine_FCVT03		:= 0.0;
		Calcul_Debit_Bypass 								:= LIMIT(0.0, 600.0 - (Consigne_Mode_EnFctnmnt_GD + Consigne_Mode_EnFctnmnt_PD), 579.0);
		GVL_RegTROX.ConsAppliDeb_Reg_Bypass_FCVT04			:= Calcul_Debit_Bypass;
		GVL_RegTROX.ConsAppliDeb_RegSouf_CabGD_FCVT05		:= Consigne_Mode_EnFctnmnt_GD;
		GVL_RegTROX.ConsAppliDeb_RegSouf_CabPD_FCVT06		:= 0.0;
		(*IF (ACH_Mode_Auto_Out_Debit_Souf < 354.0) //Mettre la valeur maximum du débit du registre en diam 100mm
			THEN
			GVL_RegTROX.ConsAppliDeb_RegSouf_CabGD_FCVT05	:= 0.0;
			GVL_RegTROX.ConsAppliDeb_RegSouf_CabPD_FCVT06	:= ACH_Mode_Auto_Out_Debit_Souf;
			ELSE
			GVL_RegTROX.ConsAppliDeb_RegSouf_CabGD_FCVT05	:= ACH_Mode_Auto_Out_Debit_Souf;
			GVL_RegTROX.ConsAppliDeb_RegSouf_CabPD_FCVT06	:= 0.0;	
		END_IF*)
		GVL_RegTROX.ConsAppliDeb_RegRep_FCVT07				:= LIMIT(0, Consigne_Mode_EnFctnmnt_GD - Consigne_Mode_EnFctnmnt_PD, 1020.0);
	ELSE // gestion sans CTA (Activation des redistres de soufflage générale uniquement et ouverture du registre FCVT03)
		IF (Cons_Deb_Soufflage_Appli < 354.0) //Mettre la valeur maximum du débit du registre en diam 100mm
			THEN
			GVL_RegTROX.ConsAppliDeb_RegSouf_GD_FCVT01		:= 0.0;
			GVL_RegTROX.ConsAppliDeb_RegSouf_PD_FCVT02		:= Cons_Deb_Soufflage_Appli;
			ELSE
			GVL_RegTROX.ConsAppliDeb_RegSouf_GD_FCVT01		:= Cons_Deb_Soufflage_Appli;
			GVL_RegTROX.ConsAppliDeb_RegSouf_PD_FCVT02		:= 0.0;	
		END_IF
		GVL_RegTROX.ConsAppliDeb_RegSouf_Cabine_FCVT03		:= 1020.0; //Mettre le débit maximum pour qu'il reste ouvert à 100%
		GVL_RegTROX.ConsAppliDeb_Reg_Bypass_FCVT04			:= 0.0;
		GVL_RegTROX.ConsAppliDeb_RegSouf_CabGD_FCVT05		:= 0.0;
		GVL_RegTROX.ConsAppliDeb_RegSouf_CabPD_FCVT06		:= 0.0;
		GVL_RegTROX.ConsAppliDeb_RegRep_FCVT07				:= 0.0;
	END_IF
END_IF;

(**********************************************Gestion de la consigne de température, de débit soufflage et de débit extraction en etat cabine nettoyage vol/h*)
IF(Mode_Cabine_Nettoyage)
	THEN
	Cons_Actionneur_Registre_Ext_Volh := Cons_Deb_Souf_Etat_Nettoyage;
	Cons_Actionneur_Registre_Souf_Volh := Cons_Deb_Souf_Etat_Nettoyage;
END_IF;

(**********************************************Gestion de la consigne de température, de débit soufflage et de débit extraction en etat cabine evaluation vol/h*)
IF(Mode_Evaluation)
	THEN
	Cons_Actionneur_Registre_Ext_Volh := Cons_Deb_Souf_Etat_Evaluation;
	Cons_Actionneur_Registre_Souf_Volh := Cons_Deb_Souf_Etat_Evaluation;
END_IF;

(**********************************************Consigne de la vanne 3 voies eau mitigée*)
(*Deux types de gestion, une via la regul PID si une vanne d'alimentation est ouverte et la deuxième si il y'a la NEP (Position de régulation au repos)*)
Mode_NEP_Chaud := Mode_Auto.Mode_18 OR Mode_Manu.Mode_18;
Mode_NEP_Froid := Mode_Auto.Mode_19 OR Mode_Manu.Mode_19;

IF(Mode_NEP_Chaud OR Mode_NEP_Froid)
	THEN
	Cons_Actionneur_V3V_Eau_Mitig := MAX(Mode_Auto.Out_Cons_V3V_Eau_Mitig , Mode_Manu.Out_Cons_V3V_Eau_Mitig);
	ELSE
	Cons_Actionneur_V3V_Eau_Mitig := S_Cmd_PID_Temp_Eau_Mitig;
END_IF;

(**********************************************Forçage ouverture electrovanne lavabo et douche pour eviter l'achéssement*******************************************************************************)
IF((Mode_Cabine_Libre AND Option_Cabine_Humide AND ((VDayOfWeek = Cons_J_Forc_Vid_Lavabo) AND (Vheure = Cons_H_Forc_Vid_Lavabo) AND (Vminute = Cons_M_Forc_Vid_Lavabo))))
	THEN
	Forc_Ouv_Alim_Lav_Dou := FALSE;
	ELSE
	Forc_Ouv_Alim_Lav_Dou := FALSE;
END_IF;

(**********************************************Convertion en m3/h pour la consigne de soufflage et d'extraction******************************************)
Cons_Actionneur_Registre_Ext_m3h := (Cons_Actionneur_Registre_Ext_Volh * Volume_Cabine);
Cons_Actionneur_Registre_Souf_m3h := (Cons_Actionneur_Registre_Souf_Volh * Volume_Cabine);

(**********************************************Convertion en °F pour la consigne de la vanne thermo******************************************)
Calcul_Temp1 := ((1.8 * Cons_Temperature_Eau) + 32.0);
Cons_Temperature_Eau_F := REAL_TO_INT(Calcul_Temp1 * 10);

(**********************************************Consigne appliquée sur le registre étanche d'extraction******************************************)
IF (Option_Reg_Etanche_Ext)
	THEN
	IF(Option_Regul_Deb_Ou_Press)
		THEN
		Cons_Actionneur_Reg_Etanche_Ext := S_Cmd_PID_Press_Cab;
		ELSE
		IF((Cons_Actionneur_Registre_Ext_m3h > ((Cons_Max_Bas_Deb_Ext + 0.5) * Volume_Cabine)))
			THEN
			Cons_Actionneur_Reg_Etanche_Ext := 100.0;
			ELSE
			Cons_Actionneur_Reg_Etanche_Ext := 0.0;
		END_IF;
	END_IF;
ELSE
	Cons_Actionneur_Reg_Etanche_Ext := 0.0;
END_IF;

(**********************************************Gestion de la consigne de débit en mode post ventilation*)
IF(Dmd_Post_Ventilation)
	THEN
	Cons_Actionneur_Registre_Ext_Volh 					:= 0.0;
	Cons_Actionneur_Registre_Souf_Volh 					:= 0.0;
	
	GVL_RegTROX.ConsAppliDeb_RegSouf_GD_FCVT01			:= 675.0;
	GVL_RegTROX.ConsAppliDeb_RegSouf_PD_FCVT02			:= 0.0;
	GVL_RegTROX.ConsAppliDeb_RegSouf_Cabine_FCVT03		:= 0.0;
	GVL_RegTROX.ConsAppliDeb_Reg_Bypass_FCVT04			:= 0.0;
	GVL_RegTROX.ConsAppliDeb_RegSouf_CabGD_FCVT05		:= 675.0;
	GVL_RegTROX.ConsAppliDeb_RegSouf_CabPD_FCVT06		:= 0.0;
	GVL_RegTROX.ConsAppliDeb_RegRep_FCVT07				:= 0.0;
END_IF;

(**********************************************Déclaration des VAV en communication******************************************)
(**********************************************VAV FCVT01*)
(*Sonde*)
GVL_RegTROX.MES_RegSouf_GD_FCVT01(
	Enable_Alarme:= TRUE, 
	Status_DEF_EAN:= GVL_RegTROX.RegSouf_GD_FCVT01_DefCom OR GVL_RegTROX.RegSouf_GD_FCVT01_Def_DiscordDeb, 
	Tempo_AL:= T#10S, 
	EAN_MIN:= 0.0, 
	EAN_MAX:= 1020.0, 
	MES_MIN:= 0.0, 
	MES_MAX:= 1020.0, 
	Filtre_Actif:= FALSE, 
	Temps_Echantillonage:= T#500MS, 
	Tab_Sonde:= GVL_RegTROX.TAB_Sonde_RegSouf_GD_FCVT01);
(*Registre*)	
GVL_RegTROX.RegSouf_GD_FCVT01(
	Cons_Pos_Dem:= GVL_RegTROX.Com_RegSouf_GD_FCVT01.MES_Pos, 
	Type_Consigne:= TRUE, 
	Control_Discordance:= FALSE, 
	Presence_Fdc:= 0, 
	Inverse_SAN:= FALSE, 
	SAN_MIN:= 0.0, 
	SAN_MAX:= 1020.0,
	Tab_RegMoto:= GVL_RegTROX.TAB_Reg_RegSouf_GD_FCVT01);
	
(**********************************************VAV FCVT02*)
(*Sonde*)
GVL_RegTROX.MES_RegSouf_PD_FCVT02(
	Enable_Alarme:= TRUE, 
	Status_DEF_EAN:= GVL_RegTROX.RegSouf_PD_FCVT02_DefCom OR GVL_RegTROX.RegSouf_PD_FCVT02_Def_DiscordDeb, 
	Tempo_AL:= T#10S, 
	EAN_MIN:= 0.0, 
	EAN_MAX:= 364.0, 
	MES_MIN:= 0.0, 
	MES_MAX:= 364.0, 
	Filtre_Actif:= FALSE, 
	Temps_Echantillonage:= T#500MS, 
	Tab_Sonde:= GVL_RegTROX.TAB_Sonde_RegSouf_PD_FCVT02);
(*Registre*)	
GVL_RegTROX.RegSouf_PD_FCVT02(
	Cons_Pos_Dem:= GVL_RegTROX.Com_RegSouf_PD_FCVT02.MES_Pos, 
	Type_Consigne:= TRUE, 
	Control_Discordance:= FALSE, 
	Presence_Fdc:= 0, 
	Inverse_SAN:= FALSE, 
	SAN_MIN:= 0.0, 
	SAN_MAX:= 364.0,
	Tab_RegMoto:= GVL_RegTROX.TAB_Reg_RegSouf_PD_FCVT02);

(**********************************************VAV FCVT03*)
(*Sonde*)
GVL_RegTROX.MES_RegSouf_Cabine_FCVT03(
	Enable_Alarme:= TRUE, 
	Status_DEF_EAN:= GVL_RegTROX.RegSouf_Cabine_FCVT03_DefCom, 
	Tempo_AL:= T#10S, 
	EAN_MIN:= 0.0, 
	EAN_MAX:= 1020.0, 
	MES_MIN:= 0.0, 
	MES_MAX:= 1020.0, 
	Filtre_Actif:= FALSE, 
	Temps_Echantillonage:= T#500MS, 
	Tab_Sonde:= GVL_RegTROX.TAB_Sonde_RegSouf_Cabine_FCVT03);
(*Registre*)	
GVL_RegTROX.RegSouf_Cabine_FCVT03(
	Cons_Pos_Dem:= GVL_RegTROX.Com_RegSouf_Cabine_FCVT03.MES_Pos, 
	Type_Consigne:= TRUE, 
	Control_Discordance:= FALSE, 
	Presence_Fdc:= 0, 
	Inverse_SAN:= FALSE, 
	SAN_MIN:= 0.0, 
	SAN_MAX:= 1020.0,
	Tab_RegMoto:= GVL_RegTROX.TAB_Reg_RegSouf_Cabine_FCVT03);

(**********************************************VAV FCVT04*)
(*Sonde*)
GVL_RegTROX.MES_RegBypass_FCVT04(
	Enable_Alarme:= TRUE, 
	Status_DEF_EAN:= GVL_RegTROX.Reg_Bypass_FCVT04_DefCom OR GVL_RegTROX.Reg_Bypass_FCVT04_Def_DiscordDeb, 
	Tempo_AL:= T#10S, 
	EAN_MIN:= 0.0, 
	EAN_MAX:= 579.0, 
	MES_MIN:= 0.0, 
	MES_MAX:= 579.0, 
	Filtre_Actif:= FALSE, 
	Temps_Echantillonage:= T#500MS, 
	Tab_Sonde:= GVL_RegTROX.TAB_Sonde_RegBypass_FCVT04);
(*Registre*)	
GVL_RegTROX.RegBypass_FCVT04(
	Cons_Pos_Dem:= GVL_RegTROX.Com_Reg_Bypass_FCVT04.MES_Pos, 
	Type_Consigne:= TRUE, 
	Control_Discordance:= FALSE, 
	Presence_Fdc:= 0, 
	Inverse_SAN:= FALSE, 
	SAN_MIN:= 0.0, 
	SAN_MAX:= 579.0,
	Tab_RegMoto:= GVL_RegTROX.TAB_Reg_RegBypass_FCVT04);
	
(**********************************************VAV FCVT05*)
(*Sonde*)
GVL_RegTROX.MES_RegSouf_CabGD_FCVT05(
	Enable_Alarme:= TRUE, 
	Status_DEF_EAN:= GVL_RegTROX.RegSouf_CabGD_FCVT05_DefCom OR GVL_RegTROX.RegSouf_CabGD_FCVT05_Def_DiscordDeb, 
	Tempo_AL:= T#10S, 
	EAN_MIN:= 0.0, 
	EAN_MAX:= 1020.0, 
	MES_MIN:= 0.0, 
	MES_MAX:= 1020.0, 
	Filtre_Actif:= FALSE, 
	Temps_Echantillonage:= T#500MS, 
	Tab_Sonde:= GVL_RegTROX.TAB_Sonde_RegSouf_CabGD_FCVT05);
(*Registre*)	
GVL_RegTROX.RegSouf_CabGD_FCVT05(
	Cons_Pos_Dem:= GVL_RegTROX.Com_RegSouf_CabGD_FCVT05.MES_Pos, 
	Type_Consigne:= TRUE, 
	Control_Discordance:= FALSE, 
	Presence_Fdc:= 0, 
	Inverse_SAN:= FALSE, 
	SAN_MIN:= 0.0, 
	SAN_MAX:= 1020.0,
	Tab_RegMoto:= GVL_RegTROX.TAB_Reg_RegSouf_CabGD_FCVT05);
	
(**********************************************VAV FCVT06*)
(*Sonde*)
GVL_RegTROX.MES_RegSouf_CabPD_FCVT06(
	Enable_Alarme:= TRUE, 
	Status_DEF_EAN:= GVL_RegTROX.RegSouf_CabPD_FCVT06_DefCom OR GVL_RegTROX.RegSouf_CabPD_FCVT06_Def_DiscordDeb, 
	Tempo_AL:= T#10S, 
	EAN_MIN:= 0.0, 
	EAN_MAX:= 364.0, 
	MES_MIN:= 0.0, 
	MES_MAX:= 364.0, 
	Filtre_Actif:= FALSE, 
	Temps_Echantillonage:= T#500MS, 
	Tab_Sonde:= GVL_RegTROX.TAB_Sonde_RegSouf_CabPD_FCVT06);
(*Registre*)	
GVL_RegTROX.RegSouf_CabPD_FCVT06(
	Cons_Pos_Dem:= GVL_RegTROX.Com_RegSouf_CabPD_FCVT06.MES_Pos, 
	Type_Consigne:= TRUE, 
	Control_Discordance:= FALSE, 
	Presence_Fdc:= 0, 
	Inverse_SAN:= FALSE, 
	SAN_MIN:= 0.0, 
	SAN_MAX:= 364.0,
	Tab_RegMoto:= GVL_RegTROX.TAB_Reg_RegSouf_CabPD_FCVT06);
	
(**********************************************VAV FCVT07*)
(*Sonde*)
GVL_RegTROX.MES_RegRep_FCVT07(
	Enable_Alarme:= TRUE, 
	Status_DEF_EAN:= GVL_RegTROX.RegRep_FCVT07_DefCom, 
	Tempo_AL:= T#10S, 
	EAN_MIN:= 0.0, 
	EAN_MAX:= 1020.0, 
	MES_MIN:= 0.0, 
	MES_MAX:= 1020.0, 
	Filtre_Actif:= FALSE, 
	Temps_Echantillonage:= T#500MS, 
	Tab_Sonde:= GVL_RegTROX.TAB_Sonde_RegRep_FCVT07);
(*Registre*)	
GVL_RegTROX.RegRep_FCVT07(
	Cons_Pos_Dem:= GVL_RegTROX.Com_RegRep_FCVT07.MES_Pos, 
	Type_Consigne:= TRUE, 
	Control_Discordance:= FALSE, 
	Presence_Fdc:= 0, 
	Inverse_SAN:= FALSE, 
	SAN_MIN:= 0.0, 
	SAN_MAX:= 1020.0,
	Tab_RegMoto:= GVL_RegTROX.TAB_Reg_RegRep_FCVT07);

END_PROGRAM

// ---- POUs/q_Gestion_Actionneurs_ANA.TcPOU
PROGRAM q_Gestion_Actionneurs_ANA
VAR
	Moteur_Aerobox_Bas_Deb: Moteur_EC;
	Batterie_Electrique: BatElec;
	Moteur_By_Pass: Moteur_EC;
	Reg_Etanche_Ext: Registre_V1;
	V3V_Eau_Mitig: Registre_V1;
END_VAR
VAR // added by the converter: edge detectors and wires of the graphical bodies
    _w1 : BOOL;
END_VAR

Cons_Actio_Registre_Ext_m3h := SEL(Enable_PID_Bas_Deb_Ext OR Arret_Extraction OR Defaut_Sonde_Press_Cabine, Cons_Actionneur_Registre_Ext_m3h, 0.0);
FCV_01_extraction(
    Enable := Option_RegExt_Ultrason,
    Type_Consigne := TRUE,
    Mode_Vidange := FALSE,
    Cons_Pos_Dem := Cons_Actio_Registre_Ext_m3h,
    Cmd_Ouv_Dem := FALSE,
    Info_Mes_Pos := 0.0,
    Presence_Fdc := 0,
    Info_Fdc_Ouvert := FALSE,
    Info_Fdc_Ferme := FALSE,
    Secu_Niveau_Haut := FALSE,
    Control_Discrodance := FALSE,
    Hyst_Al_Discord := 0.0,
    Tempo_Discord_TOR := T#0s,
    EF_Forcage := EF_Cons_Registre_Extraction,
    F_STOR_Registre := FALSE,
    F_SAN_Registre := F_Cons_Registre_Extraction,
    In_SCL_MIN_REAL := 0.0,
    In_SCL_OUT_REAL := 300.0,
    SAN_MIN := 0.0,
    SAN_MAX := 32767.0); // Registre_V1
S_Cons_Registre_Extraction := FCV_01_extraction.SAN_Cons_Registre;
Cons_Actio_Registre_Souf_m3h := SEL(Enable_PID_Bas_Deb_Ext OR Arret_Soufflage OR Defaut_Sonde_Press_Cabine, Cons_Actionneur_Registre_Souf_m3h, 0.0);
FCV_02_soufflage(
    Enable := Option_RegSouf_Ultrason,
    Type_Consigne := TRUE,
    Mode_Vidange := FALSE,
    Cons_Pos_Dem := Cons_Actio_Registre_Souf_m3h,
    Cmd_Ouv_Dem := FALSE,
    Info_Mes_Pos := 0.0,
    Presence_Fdc := 0,
    Info_Fdc_Ouvert := FALSE,
    Info_Fdc_Ferme := FALSE,
    Secu_Niveau_Haut := FALSE,
    Control_Discrodance := FALSE,
    Hyst_Al_Discord := 0.0,
    Tempo_Discord_TOR := T#0s,
    EF_Forcage := EF_Cons_Registre_Soufflage,
    F_STOR_Registre := FALSE,
    F_SAN_Registre := F_Cons_Registre_Soufflage,
    In_SCL_MIN_REAL := 0.0,
    In_SCL_OUT_REAL := 300.0,
    SAN_MIN := 0.0,
    SAN_MAX := 32767.0); // Registre_V1
S_Cons_Registre_Soufflage := FCV_02_soufflage.SAN_Cons_Registre;
Moteur_Aerobox_Bas_Deb(
    Enable := Option_Bas_Debit,
    Cons_Vit_Dem := Cons_Actionneur_Moteur_BasDebit,
    Cmd_Ma_Dem := Cons_Actionneur_Moteur_BasDebit > 5.0,
    Pres_Mes_Freq := FALSE,
    Freq_Min := 0.0,
    Freq_Max := 100.0,
    Info_Marche := FALSE,
    Info_Defaut := FALSE,
    ModeOccupe := FALSE,
    Sel_Cons_Fixe := FALSE,
    Inverse_SAN := FALSE,
    SAN_MIN := 0.0,
    SAN_MAX := 32767.0,
    Tab_Var := Tab_Mot_Aerobox_Bas_Deb); // Moteur_EC
S_Cons_Moteur_BasDebit := Moteur_Aerobox_Bas_Deb.SAN_CONS_VAR;
_w1 := Tab_MES_Sonde_Gros_Debit_Soufflage.R_MesCor > 35.0;
Batterie_Electrique(
    Enable := Option_Batt_Elec,
    Cons_BatElec_Dem := Cons_Actionneur_BattElec,
    Mes_Temp := Tab_MES_Sonde_Temp_Amb.R_MesCor,
    Info_Defaut := E_Info_Klixon_BattElec,
    Info_Ma_Mot := _w1,
    Info_Press_Sec := _w1,
    Type_Commande := TRUE,
    Inverse_SAN := FALSE,
    SAN_MIN := 0.0,
    SAN_MAX := 32767.0,
    Tab_BatElec := Tab_Batterie_Elec); // BatElec
S_Cons_BattElec := Batterie_Electrique.SAN_CONS_BAT_ELEC;
S_Cmd_BattElec := Batterie_Electrique.STOR_CMD_BAT_ELEC;
Moteur_By_Pass(
    Enable := Option_Mot_ByPass,
    Cons_Vit_Dem := Cons_Actionneur_Moteur_ByPass,
    Cmd_Ma_Dem := Cons_Actionneur_Moteur_ByPass > 5.0,
    Pres_Mes_Freq := FALSE,
    Freq_Min := 0.0,
    Freq_Max := 100.0,
    Info_Marche := FALSE,
    Info_Defaut := FALSE,
    ModeOccupe := FALSE,
    Sel_Cons_Fixe := FALSE,
    Inverse_SAN := FALSE,
    SAN_MIN := 0.0,
    SAN_MAX := 32767.0,
    Tab_Var := Tab_Mot_ByPass); // Moteur_EC
S_Cons_Moteur_ByPass := Moteur_By_Pass.SAN_CONS_VAR;
Reg_Etanche_Ext(
    Enable := Option_Reg_Etanche_Ext,
    Type_Consigne := TRUE,
    Mode_Vidange := FALSE,
    Cons_Pos_Dem := Cons_Actionneur_Reg_Etanche_Ext,
    Cmd_Ouv_Dem := FALSE,
    Info_Mes_Pos := MES_Pos_Reg_Etanche_Ext,
    Presence_Fdc := 0,
    Info_Fdc_Ouvert := FALSE,
    Info_Fdc_Ferme := FALSE,
    Secu_Niveau_Haut := FALSE,
    Defaut_Alim_Eau := FALSE,
    Control_Discrodance := TRUE,
    Hyst_Al_Discord := 10.0,
    Tempo_Discord_TOR := T#120s,
    EF_Forcage := EF_Cons_Reg_Etanche_Ext,
    F_STOR_Registre := FALSE,
    F_SAN_Registre := F_Cons_Reg_Etanche_Ext,
    In_SCL_MIN_REAL := 0.0,
    In_SCL_OUT_REAL := 100.0,
    SAN_MIN := 6553.4,
    SAN_MAX := 32767.0); // Registre_V1
S_Cons_Reg_Etanche_Ext := Reg_Etanche_Ext.SAN_Cons_Registre;
Defaut_Discord_Reg_Etanche_Ext := Reg_Etanche_Ext.Def_Discordance_ANA;
V3V_Eau_Mitig(
    Enable := Option_V3V_EauMitig,
    Type_Consigne := TRUE,
    Mode_Vidange := FALSE,
    Cons_Pos_Dem := Cons_Actionneur_V3V_Eau_Mitig,
    Cmd_Ouv_Dem := FALSE,
    Info_Mes_Pos := Cons_Actionneur_V3V_Eau_Mitig,
    Presence_Fdc := 0,
    Info_Fdc_Ouvert := FALSE,
    Info_Fdc_Ferme := FALSE,
    Secu_Niveau_Haut := FALSE,
    Defaut_Alim_Eau := FALSE,
    Control_Discrodance := FALSE,
    Hyst_Al_Discord := 10.0,
    Tempo_Discord_TOR := T#120s,
    EF_Forcage := EF_Cons_V3V_Eau_Mitig,
    F_STOR_Registre := FALSE,
    F_SAN_Registre := F_Cons_V3V_Eau_Mitig,
    In_SCL_MIN_REAL := 0.0,
    In_SCL_OUT_REAL := 100.0,
    SAN_MIN := 6553.4,
    SAN_MAX := 32767.0); // Registre_V1
S_Cons_Ouv_V3V_Eau_Mitig := V3V_Eau_Mitig.SAN_Cons_Registre;

END_PROGRAM

// ---- POUs/Block/Objets/Moteur_EC.TcPOU
FUNCTION_BLOCK Moteur_EC
VAR_INPUT
	Enable			:BOOL; (*Activation de l'objet*)
	Cons_Vit_Dem	:REAL; (*Consigne variateur demandé (venant de la Régulation) / en %*)
	Cmd_Ma_Dem	:BOOL; (*Commande marche variateur demandé (venant de la Régulation) / 1 = Marche*)
	Pres_Mes_Freq	:BOOL; (*Présence de la mesure fréquence (si pas de mesure la mesure fréquence sera calculé par LE bloc) / 1 = Présent / 0 = Absent*)
	Info_Freq		:REAL; (*Info fréquence variateur / en Hz*)
	Freq_Min		:REAL; (*Fréquence MIN variateur / en Hz*)
	Freq_Max		:REAL; (*Fréquence MAX variateur / en Hz*)
	Info_Marche		:BOOL; (*Info marche variateur (recopie ETOR) / 1 = Marche*)
	Info_Defaut		:BOOL; (*Info défaut variateur (recopie ETOR) / 1 = Défaut*)
	ModeOccupe		:BOOL; (*Mode occupé / inoccupé / 1 = Occupé / 0 = Inoccupé*)
	Sel_Cons_Fixe	:BOOL; (*Selection consigne fixe ou variable / 1 = Fixe / 0 = Variable*)
	Inverse_SAN		:BOOL; (*Inversion de la sortie SAN / 1 = Sens inverse / 0 = Sens normal*)
	SAN_MIN		:REAL; (*Valeur minimal de la sortie SAN / en point automate*)
	SAN_MAX		:REAL; (*Valeur maximal de la sortie SAN / en point automate*)
END_VAR

VAR_OUTPUT
	SAN_CONS_VAR		:INT; (*Consigne a appliqué au variateur (pour SAN) / en %*)
	STOR_CMD_MA_VAR	:BOOL; (*Commande marche a appliqué au variateur (pour STOR) / 1 = Marche*)
	STOR_RESET_VAR	:BOOL; (*Demande reset a appliqué au variateur (pour STOR) / 1 = Reset*)
END_VAR

VAR
	CONS_INT_VAR	:REAL;
	Cmd_Ma_Int	:BOOL;
	CONS_VAR	:REAL;
	Mes_Freq	:REAL;
	val_01	:REAL;
	val_02	:REAL;
	val_x	:REAL;
	val_b	:REAL;
	val_a	:REAL;
	val_y	:REAL;
	val_final	:REAL;
	val_0x	:REAL;
	val_0b	:REAL;
	val_0a	:REAL;
	val_0y	:REAL;
	Val_Calcul1	:REAL;
END_VAR

VAR_IN_OUT
	Tab_Var	:Objet_Moteur_EC; (*Tableau des valeurs*)
END_VAR

(* Gestion consigne **************************************************************)
IF Tab_Var.Mot_Ecriture.0
	THEN
		CONS_INT_VAR := Tab_Var.W_ConsForcage;
		Cmd_Ma_Int := Tab_Var.Mot_Ecriture.1;
	ELSE
		IF Cmd_Ma_Dem
			THEN
				IF Tab_Var.Mot_Lecture.4 (* Gestion consigne fixe *)
					THEN
						IF Tab_Var.Mot_Lecture.3
							THEN
								CONS_INT_VAR := Tab_Var.W_ConsOccupe;
							ELSE
								CONS_INT_VAR := Tab_Var.W_ConsInoccupe;
						END_IF;
					ELSE (* Gestion consigne varaible *)
						CONS_INT_VAR := Cons_Vit_Dem;
				END_IF;
			ELSE
				CONS_INT_VAR := 0.0;
		END_IF;
		Cmd_Ma_Int := Cmd_Ma_Dem;
END_IF;
CONS_VAR := LIMIT(Tab_Var.W_LimiteMinCons,CONS_INT_VAR,Tab_Var.W_LimiteMaxCons);


(* Gestion mesure fréquence **************************************************************)
IF Pres_Mes_Freq
	THEN
		Mes_Freq := Info_Freq;
	ELSE
		(* Mise à l'échelle de la fréquence *)
		val_01 := Freq_Max - Freq_Min;
		val_02 := Tab_Var.W_LimiteMaxCons - Tab_Var.W_LimiteMinCons;
		val_0x := CONS_VAR;
		val_0a := val_01 / MAX(1.0,val_02);
		val_0b := Freq_Max - (val_0a * Tab_Var.W_LimiteMaxCons);
		val_0y := (val_0a * val_0x) + val_0b;
		Mes_Freq := val_0y;
END_IF;
Tab_Var.R_InfoFreq := LIMIT(Freq_Min,Mes_Freq,Freq_Max);


(* Gestion sortie analogique **************************************************************)
(* Mise à l'echelle sortie ****)
val_x := CONS_VAR;
val_b := SAN_Max - (val_a * 100.0);
val_a := (SAN_Max - SAN_Min) / 100.0;
val_y := (val_a * val_x) + val_b;

(* Inversion de la sortie ANA ****)
IF (Enable)
	THEN
	IF (Inverse_SAN)
		THEN
			val_final := SAN_Max - val_y;
		ELSE
			val_final := val_y;
	END_IF;
	Val_Calcul1 := LIMIT(SAN_Min,val_final, SAN_Max);
	SAN_CONS_VAR := REAL_TO_INT(Val_Calcul1);
	ELSE
	SAN_CONS_VAR := 0;
END_IF;


(* Gestion sortie TOR **************************************************************)
IF (Enable)
	THEN
	STOR_CMD_MA_VAR := Cmd_Ma_Int AND NOT Info_Defaut;
	STOR_RESET_VAR 	:= Tab_Var.Mot_Ecriture.2;
	ELSE
	STOR_CMD_MA_VAR := FALSE;
	STOR_RESET_VAR 	:= FALSE;
END_IF;

(* Recopie pour lecture GTC *********************************************************)
Tab_Var.Mot_Lecture.0			:= STOR_CMD_MA_VAR;
Tab_Var.Mot_Lecture.1			:= Info_Defaut;
Tab_Var.Mot_Lecture.2			:= STOR_CMD_MA_VAR;
Tab_Var.Mot_Lecture.3			:= ModeOccupe;
Tab_Var.Mot_Lecture.4			:= Sel_Cons_Fixe;

Tab_Var.R_LimiteMinFreq		:= Freq_Min;
Tab_Var.R_LimiteMaxFreq		:= Freq_Max;
Tab_Var.R_InfoCons			:= CONS_VAR;

END_FUNCTION_BLOCK

// ---- POUs/Block/Objets/BatElec.TcPOU
FUNCTION_BLOCK BatElec
VAR_INPUT
	Enable				:BOOL;
	Cons_BatElec_Dem	:REAL;	(*Consigne batterie éléctrique demandé (venant de la Régulation) / en %*)
	Cmd_BatElec_Dem	:BOOL;
	Mes_Temp			:REAL;	(*Mesure température apréS batterie / en °C*)
	Info_Defaut			:BOOL;	(*VAR_INPUT	Info défaut klixon batterie electrique (Recopie ETOR) / 1 = Défaut*)
	Info_Ma_Mot			:BOOL;	(*Récupération de l'information marche du moteur de ventilation*)
	Info_Press_Sec		:BOOL;	(*Récupération du pressostat de sécurité de présence d'air*)
	Type_Commande		:BOOL;	(*VAR_INPUT	Choix du TYPE de pilotage de la batterie éléctrique / 0 = PWM / 1 = ANA*)
	Inverse_SAN			:BOOL;	(*Inversion de la sortie SAN / 1 = Sens inverse / 0 = Sens normal*)
	SAN_MIN			:REAL;	(*Valeur minimal de la sortie SAN / en point automate*)
	SAN_MAX			:REAL;	(*Valeur maximal de la sortie SAN / en point automate*)
END_VAR

VAR_OUTPUT
	SAN_CONS_BAT_ELEC	:INT;	(*Consigne a appliqué à la batterie éléctrique (pour SAN) / en %*)
	STOR_CMD_BAT_ELEC	:BOOL;	(*VAR_OUTPUT	Commande a appliqué à la batterie éléctrique (pour STOR PWM) / 1 = Marche*)
	OUT_Info_Temps_Cycle	:TIME;	(*VAR_OUTPUT	Temps de cycle restant / En sec*)
END_VAR

VAR
	OUT_PWM			:BOOL;	(*Sortie du PWM / 1 = Marche*)
	Temp_ON			:REAL;
	TP_1				:TP;
	TIME_BaseTemps	:TIME;
	TIME_Temp_ON		:TIME;
	DINT_BaseTemps	:DINT;
	DINT_Temp_ON		:DINT;
	front					:BOOL;
	Temp_ON_bis		:REAL;
	TON_PWM			:TON;

	CONS_BATELEC_INT	:REAL;
	CONS_BAT_ELEC	:REAL;
	val_x				:REAL;
	val_b				:REAL;
	val_a				:REAL;
	val_y				:REAL;
	val_final				:REAL;
	Val_Calcul1			:REAL;
END_VAR

VAR_IN_OUT
	Tab_BatElec	:Objet_BatElec; (*Tableau des valeurs*)
END_VAR

(* Gestion consigne **************************************************************)
IF Tab_BatElec.Mot_Ecriture.0
	THEN
		CONS_BATELEC_INT := Tab_BatElec.W_ConsForcage;
	ELSE
		CONS_BATELEC_INT := Cons_BatElec_Dem;
END_IF;
CONS_BAT_ELEC := LIMIT(Tab_BatElec.W_LimiteMinCons,CONS_BATELEC_INT,Tab_BatElec.W_LimiteMaxCons);


(* Gestion PWM **************************************************************)
IF NOT(Type_Commande)
	THEN
		(* Cacule temps PWM *)
		Temp_ON := (Tab_BatElec.W_PeriodePWM / 100.0) * CONS_BAT_ELEC;
	
		(* Sécurité Temp On Max *)
		IF Temp_ON > Tab_BatElec.W_TempsMaxPWM
			THEN
				Temp_ON_bis := Tab_BatElec.W_TempsMaxPWM;
			ELSE
				Temp_ON_bis := Temp_ON;
		END_IF;	
		DINT_BaseTemps := REAL_TO_DINT(Tab_BatElec.W_PeriodePWM);
		TIME_BaseTemps := DINT_TO_TIME(DINT_BaseTemps * 1000);
		DINT_Temp_ON := REAL_TO_DINT(Temp_ON_bis * 10);
		TIME_Temp_ON := DINT_TO_TIME(DINT_Temp_ON * 100);

		(* Sécurité si Temps ON < Temps MIN on active pas la sortie *)
		IF (Temp_ON > Tab_BatElec.W_TempsMinPWM)
			THEN
				TP_1(IN := front,PT := TIME_Temp_ON);
				OUT_PWM := TP_1.Q;
			ELSE
				OUT_PWM := FALSE;
		END_IF;
		IF CONS_BAT_ELEC = 0.0
			THEN
				OUT_PWM := FALSE;
		END_IF;
		IF ((CONS_BAT_ELEC = 100.0) AND (Temp_ON = Tab_BatElec.W_TempsMaxPWM))
			THEN
				OUT_PWM := TRUE;
		END_IF;

		TON_PWM(IN := TRUE AND NOT(TON_PWM.Q), PT := TIME_BaseTemps);
		front := TON_PWM.Q;
		OUT_Info_Temps_Cycle := TON_PWM.ET;
	ELSE
		OUT_PWM := FALSE;
		OUT_Info_Temps_Cycle := t#0s;
END_IF;


(* Gestion sortie analogique ou TOR **************************************************************)
IF Type_Commande
	THEN (* Gestion sortie analogique *)
		(* Mise à l'echelle sortie ****)
		val_x := CONS_BAT_ELEC;
		val_b := SAN_Max - (val_a * 100.0);
		val_a := (SAN_Max - SAN_Min) / 100.0;
		val_y := (val_a * val_x) + val_b;

		(* Inversion de la sortie ANA ****)
		IF (Inverse_SAN)
			THEN
				val_final := SAN_Max - val_y;
			ELSE
				val_final := val_y;
		END_IF;
		Val_Calcul1 := LIMIT(SAN_Min,val_final, SAN_Max);
		SAN_CONS_BAT_ELEC := REAL_TO_INT(Val_Calcul1);
		STOR_CMD_BAT_ELEC := Cmd_BatElec_Dem AND Info_Ma_Mot AND Info_Press_Sec AND Info_Defaut;
	ELSE (* Gestion sortie TOR PWM *)
		SAN_CONS_BAT_ELEC := 0;
		STOR_CMD_BAT_ELEC :=  OUT_PWM AND Info_Ma_Mot AND Info_Press_Sec AND Info_Defaut;
END_IF;

IF(NOT Enable)
	THEN
	CONS_BAT_ELEC := 0.0;
	SAN_CONS_BAT_ELEC := 0;
	STOR_CMD_BAT_ELEC := FALSE;
END_IF;

(* Recopie pour lecture GTC *********************************************************)
Tab_BatElec.Mot_Lecture.0	:= 	STOR_CMD_BAT_ELEC;
Tab_BatElec.Mot_Lecture.1	:= 	Info_Defaut;
Tab_BatElec.Mot_Lecture.2	:= 	Type_Commande;
Tab_BatElec.R_Info_Cons		:= 	CONS_BAT_ELEC;
Tab_BatElec.R_TempApresBat	:= 	Mes_Temp;

(* Recopie pour lecture GTC *********************************************************)
Tab_BatElec.Mot_Lecture.0	:= 	STOR_CMD_BAT_ELEC;
Tab_BatElec.Mot_Lecture.1	:= 	Info_Defaut;
Tab_BatElec.Mot_Lecture.2	:= 	Type_Commande;
Tab_BatElec.R_Info_Cons		:= 	CONS_BAT_ELEC;
Tab_BatElec.R_TempApresBat	:= 	Mes_Temp;

END_FUNCTION_BLOCK

// ---- POUs/Block/Cabines/Registre_V1.TcPOU
FUNCTION_BLOCK Registre_V1
VAR_INPUT
	Enable:					BOOL;	(*Mise en route du bloc de fonction*)
	Type_Consigne:			BOOL;	 (*Choix du type de pilotage du registre / 1 = ANA / 0 = TOR*)
	Mode_Vidange:			BOOL; 	(*Mode de vidange / 1=Mode vidange / 0= Mode alimentation douche, Douchette, Lavabo, etc...*)
	Cons_Pos_Dem:			REAL; 	(*Consigne position registre demandé (Venant de la régulation) / en %*)
	Cmd_Ouv_Dem:			BOOL; 	(*Commande ouverture registre demandé (Venant de la régulation) / 1 = Ouverture*)
	Info_Mes_Pos:			REAL; 	(*Info mesure position registre (recopie EAN) / en %*)
	Presence_Fdc:			INT; 	(*Mot de présence des fin de course / 0 = Pas de fin de course / 1 = Fin de course Ouvert / 2 = Fin de course Fermé / 3 = Les 2 fin de course*)
	Info_Fdc_Ouvert:			BOOL; 	(*Info fin de course ouvert (recopie ETOR) / 1 = Ouvert*)
	Info_Fdc_Ferme:			BOOL; 	(*Info fin de course fermé (recopi ETOR) / 1 = Fermé*)
	Secu_Niveau_Haut:		BOOL; 	(*Sécurité du niveau haut / 0 = Niveau haut actif*)
	Defaut_Alim_Eau:			BOOL;	(*Sécurité qui coupe l'alimentation en eau*)
	Control_Discrodance:		BOOL;	 (*Autorisation de marche des alarmes / 1 = Alarme autorisé*)
	Hyst_Al_Discord:			REAL;	 (*Hystéresis pour le défaut discordance en type ANA*)
	Tempo_Discord_TOR:		TIME; 	(*Temporisation du défaut discordance en type TOR*)
	EF_Forcage:				BOOL;	 (*Enable forçage du registre / 1= Autorisé*)
	F_STOR_Registre: 		BOOL;	 (*Forçage du registre pour le mode TOR / 1= Forcé*)
	F_SAN_Registre:			REAL; 	(*Forçage du registre pour le mode ANA / en %*)
	In_SCL_MIN_REAL: REAL;
	In_SCL_OUT_REAL: REAL;
	SAN_MIN: REAL;
	SAN_MAX: REAL;
END_VAR
VAR_OUTPUT
	SAN_Cons_Registre:		INT; (*Consigne a appliqué au registre ANA (pour SAN) / en %*)
	STOR_Cmd_Ouv_Registre: BOOL; (*Commande a appliqué au registre TOR (pour STOR) / 1 = Ouverture*)
	Def_Discordance_ANA:BOOL;
	Def_Discordance_Ouverture:BOOL;
	Def_Discordance_Fermeture: BOOL;
END_VAR
VAR
	Cons_Registre:			REAL;
	iCons_Registre:			INT;
	Cmd_Registre:			BOOL;
	SCL_ANA: 				SCL;
	TON_1:					TON;
	TON_2:					TON;
	TON_3:					TON;
	TON_4:					TON;
	TON_5:					TON;
	TON_6:					TON;
	RS_1:					RS;
	RS_2:					RS;
	Calcul_1: REAL;
	Calcul_2: REAL;
END_VAR

IF(Enable)
	THEN
	(*======================Gestion de la Consigne===================================*)
	IF(Type_Consigne)
		THEN			(* Gestion consigne pour un registre ANA *)
		Cmd_Registre := FALSE;
		IF(EF_Forcage)
			THEN
				Cons_Registre := F_SAN_Registre;
			ELSE
				Cons_Registre := Cons_Pos_Dem;
		END_IF;
	ELSE				 (* Gestion consigne pour un registre TOR *)
		Cons_Registre := 0.0;
		IF(EF_Forcage)
			THEN
				Cmd_Registre := F_STOR_Registre;
			ELSE
				Cmd_Registre := Cmd_Ouv_Dem;
		END_IF
	END_IF;
	
	(*======================Gestion de la sortie Analogique==============================*)
	iCons_Registre := REAL_TO_INT(Cons_Registre); (*Convertion de la consigne analogique*)
	SCL_ANA(
		IN_INT:= iCons_Registre,
		LIM_MIN_IN_REAL:= In_SCL_MIN_REAL,
		LIM_MAX_IN_REAL:= In_SCL_OUT_REAL,
		LIM_MIN_OUT_REAL:= SAN_MIN,(*0V*)
		LIM_MAX_OUT_REAL:= SAN_MAX,(*10V*)
		OUT_INT=> SAN_Cons_Registre);
	
	(*======================Gestion de la sortie TOR====================================*)
	IF( Mode_Vidange)
		THEN (*Gestion de la STOR en fonction du mode de vidange*)
		IF(Secu_Niveau_Haut)
			THEN
				STOR_Cmd_Ouv_Registre := TRUE;
			ELSE
				STOR_Cmd_Ouv_Registre := Cmd_Registre;
		END_IF;
	ELSE (*Gestion de la STOR en fonction du mode alimentation*)
		IF(Secu_Niveau_Haut)
			THEN
				STOR_Cmd_Ouv_Registre := FALSE;
			ELSE
				STOR_Cmd_Ouv_Registre := Cmd_Registre AND NOT Defaut_Alim_Eau;
		END_IF;
	END_IF;
	
	(*======================Gestion du défaut de discordance============================*)
	IF(Control_Discrodance)
		THEN		(*Lors du contrôle de discordance*)
			IF(Type_Consigne)
				THEN		(* Alarme discordance pour registre SAN *)
					Calcul_1 := (Cons_Registre - Hyst_Al_Discord) ;
					Calcul_2 := (Cons_Registre + Hyst_Al_Discord) ;
					TON_1(IN := ((Calcul_1 > Info_Mes_Pos) OR (Calcul_2 < Info_Mes_Pos)),PT := T#150s);
					Def_Discordance_ANA:= TON_1.Q;
			ELSE			(* Alarme discordance pour registre STOR *)
				CASE Presence_Fdc OF
					0	:	(*Mode pas de fin de course*)
							Def_Discordance_Ouverture := FALSE;
							Def_Discordance_Fermeture := FALSE;
					1	:	(*Mode Fdc ouverture uniquement*)
							TON_2(IN := ( STOR_Cmd_Ouv_Registre AND NOT Info_Fdc_Ouvert ), PT := Tempo_Discord_TOR);
							Def_Discordance_Ouverture:= TON_2.Q;
							Def_Discordance_Fermeture := FALSE;
					2	:	(*Mode Fdc fermeture uniquement*)
							TON_3(IN := ( NOT STOR_Cmd_Ouv_Registre AND NOT Info_Fdc_Ferme ), PT := Tempo_Discord_TOR);
							Def_Discordance_Fermeture:= TON_3.Q;
							Def_Discordance_Ouverture := FALSE;
					3	:	(*Mode Fdc ouverture et fermeture*)
							TON_4(IN := ((STOR_Cmd_Ouv_Registre AND NOT Info_Fdc_Ouvert)),PT := Tempo_Discord_TOR);
							TON_5(IN := ((NOT STOR_Cmd_Ouv_Registre AND NOT Info_Fdc_Ferme )),PT := Tempo_Discord_TOR);
							TON_6(IN := (Info_Fdc_Ouvert AND Info_Fdc_Ferme) ,PT := Tempo_Discord_TOR);
							RS_1(SET:= TON_4.Q, RESET1:= Info_Fdc_Ouvert);
							RS_2(SET:= TON_5.Q, RESET1:= Info_Fdc_Ferme);
							Def_Discordance_Ouverture:= RS_1.Q1 OR TON_6.Q;
							Def_Discordance_Fermeture:= RS_2.Q1 OR TON_6.Q;
	
					ELSE  (*Si Presence_Fdc > à 3*)
					Def_Discordance_Ouverture := FALSE;
					Def_Discordance_Fermeture := FALSE;
				END_CASE;
			END_IF;
		ELSE		(* Si contrôle d'alarme discordance désactivé *)
			Def_Discordance_ANA := FALSE;
			Def_Discordance_Ouverture := FALSE;
			Def_Discordance_Fermeture := FALSE;
	END_IF;
	ELSE
			SAN_Cons_Registre := 0;
			STOR_Cmd_Ouv_Registre := FALSE;
			Def_Discordance_ANA := FALSE;
			Def_Discordance_Ouverture := FALSE;
			Def_Discordance_Fermeture := FALSE;
END_IF;

END_FUNCTION_BLOCK

// ---- POUs/r_Gestion_Actionneurs_TOR.TcPOU
PROGRAM r_Gestion_Actionneurs_TOR
VAR
	XV_Alim_Douche: Registre_V1;
	XV_Alim_Douchette: Registre_V1;
	XV_Alim_Lavabo: Registre_V1;
	XV_Vid_Douche: Registre_V1;
	XV_Vid_Lavabo: Registre_V1;
	XV_Electrovanne_Douche: Registre_V1;
	XV_Electrovanne_Lavabo: Registre_V1;
	Prise_Cabine: Prise;
	XV_Vanne_Souf_Bas_Deb: Registre_V1;
	XV_Vanne_Ext_Bas_Deb: Registre_V1;
	Reg_Etanche_Souf: Registre_V1;
	XV_Alim_NEP: Registre_V1;
	Y_Verin_WC_GV: Registre_V1;
	Y_Verin_WC_PV: Registre_V1;
	Gestion_EA_WC: Sontay_4RM;
END_VAR

